	PROC WELD_20s_ALL()
        ActUnit STN1;
	    AccSet 75, 75;
	    MoveJ pjthomeSTA1zero, vCellSpeed, fine, tWeldGun\WObj:=wobj0;
        TPErase;
        !UNtilt19;
        TPWrite "NOW SEARCHING THE FIRST HALF OF WELD 'G'";
		GOTO GPOINT1stHALF;
        !!!!THIS IS THE ENTIRE "G" Search in Position EDIT STRING IN CORRECT ORDER!!!!
		PDispOff;
		MoveJ G19air2, vExtMax, z1, tWeldGun\WObj:=wobjHsideplate;
		MoveL RelTool(YG19S,0,-100,-150), v500, z1, tWeldGun\WObj:=wobjHsideplate;
		Search_1D SR_YZ_TEMP\SearchStop:=YZ_Temp, YG19S, YG19E, v300, tWeldGun\WObj:=wobjHsideplate\SchSpeed:=10;
         GHLM_YZ_POINT_SETTER G19, YZ_Temp, AA19;
        TPWrite "SRG19 XYZ:="\Pos:=SR_YZ_TEMP.trans;
		MoveL RelTool(YG19S,0,0,0), v500, z1, tWeldGun\WObj:=wobjHsideplate;
		Search_1D SR_YZ_TEMP\SearchStop:=YZ_Temp, YG15S, YG15E, v300, tWeldGun\WObj:=wobjHsideplate\SchSpeed:=10;
         GHLM_YZ_POINT_SETTER G15, YZ_Temp, AA15;
        TPWrite "SRG15 XYZ:="\Pos:=SR_YZ_TEMP.trans;
		MoveL RelTool(YG15S,0,0,0), v500, z1, tWeldGun\WObj:=wobjHsideplate;
		Search_1D SR_YZ_TEMP\SearchStop:=YZ_Temp, YG21S, YG21E, v300, tWeldGun\WObj:=wobjHsideplate\SchSpeed:=10;
         GHLM_YZ_POINT_SETTER G21, YZ_Temp, AA21;
        TPWrite "SRG21 XYZ:="\Pos:=SR_YZ_TEMP.trans;
		MoveL RelTool(YG21S,0,0,0), v500, z1, tWeldGun\WObj:=wobjHsideplate;
		Search_1D SR_YZ_TEMP\SearchStop:=YZ_Temp, YG0S, YG0E, v300, tWeldGun\WObj:=wobjHsideplate\SchSpeed:=10;
         GHLM_YZ_POINT_SETTER G0, YZ_Temp, AA0;
        TPWrite "SRG0 XYZ:="\Pos:=SR_YZ_TEMP.trans;
		MoveL RelTool(YG0S,0,0,0), v500, z1, tWeldGun\WObj:=wobjHsideplate;
		Search_1D SR_YZ_TEMP\SearchStop:=YZ_Temp, YG25S, YG25E, v300, tWeldGun\WObj:=wobjHsideplate\SchSpeed:=10;
         GHLM_YZ_POINT_SETTER G25, YZ_Temp, AA25;
        TPWrite "SRG25 XYZ:="\Pos:=SR_YZ_TEMP.trans;
		MoveL RelTool(YG25S,0,0,0), v500, z1, tWeldGun\WObj:=wobjHsideplate;
		Search_1D SR_YZ_TEMP\SearchStop:=YZ_Temp, YG29S, YG29E, v300, tWeldGun\WObj:=wobjHsideplate\SchSpeed:=10;
         GHLM_YZ_POINT_SETTER G29, YZ_Temp, AA29;
        TPWrite "SRG29 XYZ:="\Pos:=SR_YZ_TEMP.trans;
		MoveL RelTool(YG29S,0,0,0), v500, z1, tWeldGun\WObj:=wobjHsideplate;
		MoveJ G29air3, vExtMax, z1, tWeldGun\WObj:=wobjHsideplate;
        SEARCH_Gx;
        SET_G20s_X;
		PDispOff;
		MoveJ G19air1, vExtMax, z1, tWeldGun\WObj:=wobjHsideplate;
		MoveJ RelTool(G195L,0,-50,-50), v300, z1, tWeldGun\WObj:=wobjHtip;
		MoveL G195L, v100, z1, tWeldGun\WObj:=wobjHtip;
		MoveL G195, v100, z1, tWeldGun\WObj:=wobjHtip;
		MoveL G19, v100, z1, tWeldGun\WObj:=wobjHsideplate;
		MoveL RelTool(G15,0,0,-15), v100, z1, tWeldGun\WObj:=wobjHsideplate;
		MoveL G15, v100, z1, tWeldGun\WObj:=wobjHsideplate;
		MoveL RelTool(G21,0,0,-15), v100, z1, tWeldGun\WObj:=wobjHsideplate;
		MoveL G21, v100, z1, tWeldGun\WObj:=wobjHsideplate;
		MoveL RelTool(G21,0,0,-15), v100, z1, tWeldGun\WObj:=wobjHsideplate;
		MoveL G0, v100, z1, tWeldGun\WObj:=wobjHsideplate;
		MoveL RelTool(G0,0,0,-15), v100, z1, tWeldGun\WObj:=wobjHsideplate;
		MoveL RelTool(G25,0,0,-15), v100, z1, tWeldGun\WObj:=wobjHsideplate;
		MoveL G25, v100, z1, tWeldGun\WObj:=wobjHsideplate;
		MoveL RelTool(G25,0,0,-150), v100, z1, tWeldGun\WObj:=wobjHsideplate;
		MoveL G29, v100, z1, tWeldGun\WObj:=wobjHsideplate;
		MoveL RelTool(G29,0,0,-150), v100, z1, tWeldGun\WObj:=wobjHsideplate;
		MoveL RelTool(G0,0,0,-150), v100, z1, tWeldGun\WObj:=wobjHsideplate;
        !!  IF THIS IS AN H ARM THEN WE WILL RUN 1_THRU_8
        !!  IF THIS IS A G ARM THEN WE WILL RUN THE CAM-SIDE WELDS
		PDispOff;
         SET_G20s_X;
		MoveJ RelTool(G195L,0,-150,-150), v300, z1, tWeldGun\WObj:=wobjHtip;
        GOTO GWELDFIRST;
        GPOINT1stHALF:
        !!!!GETTING IN POSITION FOR THE FIRST 3 Y SEARCHES ON THE G WELD
        PDispOff;
		MoveJ G19air1, vExtMax, z1, tWeldGun\WObj:=wobjHsideplate;
		MoveL RelTool(YG19S,0,-100,-150), v500, z1, tWeldGun\WObj:=wobjHsideplate;
		Search_1D SR_YZ_TEMP\SearchStop:=YZ_Temp, YG19S, YG19E, v300, tWeldGun\WObj:=wobjHsideplate\SchSpeed:=10;
         GHLM_YZ_POINT_SETTER G19, YZ_Temp, AA19;
        TPWrite "SRG19 XYZ:="\Pos:=SR_YZ_TEMP.trans;
		MoveL RelTool(YG19S,0,0,0), v500, z1, tWeldGun\WObj:=wobjHsideplate;
		Search_1D SR_YZ_TEMP\SearchStop:=YZ_Temp, YG15S, YG15E, v300, tWeldGun\WObj:=wobjHsideplate\SchSpeed:=10;
         GHLM_YZ_POINT_SETTER G15, YZ_Temp, AA15;
        TPWrite "SRG15 XYZ:="\Pos:=SR_YZ_TEMP.trans;
		MoveL RelTool(YG15S,0,0,0), v500, z1, tWeldGun\WObj:=wobjHsideplate;
		Search_1D SR_YZ_TEMP\SearchStop:=YZ_Temp, YG21S, YG21E, v300, tWeldGun\WObj:=wobjHsideplate\SchSpeed:=10;
         GHLM_YZ_POINT_SETTER G21, YZ_Temp, AA21;
        TPWrite "SRG21 XYZ:="\Pos:=SR_YZ_TEMP.trans;
		MoveL RelTool(YG21S,0,0,0), v500, z1, tWeldGun\WObj:=wobjHsideplate;
		MoveL RelTool(YG21S,0,-100,0), v500, z1, tWeldGun\WObj:=wobjHsideplate;
 		MoveJ G19air1, vExtMax, z1, tWeldGun\WObj:=wobjHsideplate;
        SEARCH_Gx;
        SET_G20s_X;
		MoveJ G19air1, vExtMax, z1, tWeldGun\WObj:=wobjHsideplate;
		MoveJ RelTool(G195L,0,-50,-150), vExtMax, z1, tWeldGun\WObj:=wobjHtip;
        GWELDFIRST:
        IF bWO458only = TRUE OR bWO459only = TRUE THEN
        dripstop_G;
        ENDIF
        TPWrite "NOW WELDING THE FIRST THIRD OF WELD 'G'";
		MoveL RelTool(G195L,0,-50,-150), vExtMax, z1, tWeldGun\WObj:=wobjHtip;
		ArcLStart G195L, v100, smGH29, wdGH29\Weave:=wvGH29, fine, tWeldGun\WObj:=wobjHtip\Track:=trGHTBR;
		ArcL G195, v100, smGH29, wdGH29\Weave:=wvGH29, z1, tWeldGun\WObj:=wobjHtip\Track:=trGHTBR;
		ArcCEnd G15, G21, v100, smGH29, wdGH29\Weave:=wvGH29, fine, tWeldGun\WObj:=wobjHsideplate\Track:=trGHTBR;
		MoveL RelTool(G21,0,0,-150), vExtMax, z1, tWeldGun\WObj:=wobjHsideplate;
		MoveJ RelTool(G21,0,0,-200), vExtMax, z1, tWeldGun\WObj:=wobjHsideplate;
		MoveJ pjthomeSTA1zero, vCellSpeed, fine, tWeldGun\WObj:=wobj0;
        !!GOING TO THE H SIDE!!!
           MoveJ RelTool(H21,0,0,-500), vExtMax, z1, tWeldGun\WObj:=wobjHsideplate;
        TPErase;
        TPWrite "NOW WORKING ON FIRST HALF OF WELD 'H'";
		GOTO HPOINT1stHALF;
        !!!!THIS IS THE ENTIRE "H" SEARCHES EDIT STRING IN CORRECT ORDER!!!!
		PDispOff;
		MoveJ H19air1, vExtMax, z1, tWeldGun\WObj:=wobjHsideplate;
		MoveL RelTool(YH19S,150,70,-150), v500, z1, tWeldGun\WObj:=wobjHsideplate;
		Search_1D SR_YZ_TEMP\SearchStop:=YZ_Temp, YH19S, YH19E, v300, tWeldGun\WObj:=wobjHsideplate\SchSpeed:=10;
         GHLM_YZ_POINT_SETTER H19, YZ_Temp, AA19;
        TPWrite "SRH19 XYZ:="\Pos:=SR_YZ_TEMP.trans;
		MoveL RelTool(YH19S,0,0,0), v500, z1, tWeldGun\WObj:=wobjHsideplate;
		Search_1D SR_YZ_TEMP\SearchStop:=YZ_Temp, YH15S, YH15E, v300, tWeldGun\WObj:=wobjHsideplate\SchSpeed:=10;
         GHLM_YZ_POINT_SETTER H15, YZ_Temp, AA15;
        TPWrite "SRH15 XYZ:="\Pos:=SR_YZ_TEMP.trans;
		MoveL RelTool(YH15S,0,0,0), v500, z1, tWeldGun\WObj:=wobjHsideplate;
		Search_1D SR_YZ_TEMP\SearchStop:=YZ_Temp, YH21S, YH21E, v300, tWeldGun\WObj:=wobjHsideplate\SchSpeed:=10;
         GHLM_YZ_POINT_SETTER H21, YZ_Temp, AA21;
        TPWrite "SRH21 XYZ:="\Pos:=SR_YZ_TEMP.trans;
		MoveL RelTool(YH21S,0,0,0), v500, z1, tWeldGun\WObj:=wobjHsideplate;
		Search_1D SR_YZ_TEMP\SearchStop:=YZ_Temp, YH0S, YH0E, v300, tWeldGun\WObj:=wobjHsideplate\SchSpeed:=10;
         GHLM_YZ_POINT_SETTER H0, YZ_Temp, AA0;
        TPWrite "SRH0 XYZ:="\Pos:=SR_YZ_TEMP.trans;
		MoveL RelTool(YH0S,0,0,0), v500, z1, tWeldGun\WObj:=wobjHsideplate;
		Search_1D SR_YZ_TEMP\SearchStop:=YZ_Temp, YH25S, YH25E, v300, tWeldGun\WObj:=wobjHsideplate\SchSpeed:=10;
         GHLM_YZ_POINT_SETTER H25, YZ_Temp, AA25;
        TPWrite "SRH25 XYZ:="\Pos:=SR_YZ_TEMP.trans;
		MoveL RelTool(YH25S,0,0,0), v500, z1, tWeldGun\WObj:=wobjHsideplate;
		Search_1D SR_YZ_TEMP\SearchStop:=YZ_Temp, YH29S, YH29E, v300, tWeldGun\WObj:=wobjHsideplate\SchSpeed:=10;
         GHLM_YZ_POINT_SETTER H29, YZ_Temp, AA29;
        TPWrite "SRH29 XYZ:="\Pos:=SR_YZ_TEMP.trans;
		MoveL RelTool(YH29S,0,0,0), v500, z1, tWeldGun\WObj:=wobjHsideplate;
		MoveL RelTool(YH29S,100,100,0), v500, z1, tWeldGun\WObj:=wobjHsideplate;
		MoveJ H29air1, vExtMax, z1, tWeldGun\WObj:=wobjHsideplate;
        SEARCH_Hx;
        SET_H20s_X;
		MoveJ H19air1, vExtMax, z1, tWeldGun\WObj:=wobjHsideplate;
		MoveJ RelTool(H19,0,-100,-250), vExtMax, z1, tWeldGun\WObj:=wobjHsideplate;
		MoveL RelTool(H195L,0,-50,-50), v300, z1, tWeldGun\WObj:=wobjHtip;
        !!!!THIS IS THE ENTIRE "H" BASEPOINTS EDIT STRING IN CORRECT ORDER!!!!
		MoveL H195L, v100, z1, tWeldGun\WObj:=wobjHtip;
		MoveL H195, v100, z1, tWeldGun\WObj:=wobjHtip;
		MoveL H19, v100, z1, tWeldGun\WObj:=wobjHsideplate;
		MoveL RelTool(H15,0,0,-15), v100, z1, tWeldGun\WObj:=wobjHsideplate;
		MoveL H15, v100, z1, tWeldGun\WObj:=wobjHsideplate;
		MoveL RelTool(H21,0,0,-15), v100, z1, tWeldGun\WObj:=wobjHsideplate;
		MoveL H21, v100, z1, tWeldGun\WObj:=wobjHsideplate;
		MoveL RelTool(H0,0,0,-35), v100, z1, tWeldGun\WObj:=wobjHsideplate;
		MoveL H0, v100, z1, tWeldGun\WObj:=wobjHsideplate;
		MoveL RelTool(H25,0,0,-15), v100, z1, tWeldGun\WObj:=wobjHsideplate;
		MoveL H25, v100, z1, tWeldGun\WObj:=wobjHsideplate;
		MoveL RelTool(H25,0,0,-15), v100, z1, tWeldGun\WObj:=wobjHsideplate;
		MoveL H29, v100, z1, tWeldGun\WObj:=wobjHsideplate;
		MoveL RelTool(H29,0,0,-150), v100, z1, tWeldGun\WObj:=wobjHsideplate;
		MoveL RelTool(H0,0,0,-150), v100, z1, tWeldGun\WObj:=wobjHsideplate;
		PDispOff;
        PDispOff;
        SET_H20s_X;
		MoveJ RelTool(H195L,0,-150,-150), v300, z1, tWeldGun\WObj:=wobjHtip;
        GOTO HWELDSFIRSThalf;
        HPOINT1stHALF:
		PDispOff;
        !!!!GETTING IN POSITION FOR THE FIRST 3 Y SEARCHES ON THE H WELD
		MoveJ H19air1, vExtMax, z1, tWeldGun\WObj:=wobjHsideplate;
		MoveL RelTool(YH19S,150,70,-150), v500, z1, tWeldGun\WObj:=wobjHsideplate;
		Search_1D SR_YZ_TEMP\SearchStop:=YZ_Temp, YH19S, YH19E, v300, tWeldGun\WObj:=wobjHsideplate\SchSpeed:=10;
         GHLM_YZ_POINT_SETTER H19, YZ_Temp, AA19;
        TPWrite "SRH19 XYZ:="\Pos:=SR_YZ_TEMP.trans;
		MoveL RelTool(YH19S,0,0,0), v500, z1, tWeldGun\WObj:=wobjHsideplate;
		Search_1D SR_YZ_TEMP\SearchStop:=YZ_Temp, YH15S, YH15E, v300, tWeldGun\WObj:=wobjHsideplate\SchSpeed:=10;
         GHLM_YZ_POINT_SETTER H15, YZ_Temp, AA15;
        TPWrite "SRH15 XYZ:="\Pos:=SR_YZ_TEMP.trans;
		MoveL RelTool(YH15S,0,0,0), v500, z1, tWeldGun\WObj:=wobjHsideplate;
		Search_1D SR_YZ_TEMP\SearchStop:=YZ_Temp, YH21S, YH21E, v300, tWeldGun\WObj:=wobjHsideplate\SchSpeed:=10;
         GHLM_YZ_POINT_SETTER H21, YZ_Temp, AA21;
        TPWrite "SRH21 XYZ:="\Pos:=SR_YZ_TEMP.trans;
		MoveL RelTool(YH21S,0,0,0), v500, z1, tWeldGun\WObj:=wobjHsideplate;
		MoveL RelTool(YH21S,100,100,-150), v500, z1, tWeldGun\WObj:=wobjHsideplate;
        !!!!GETTING IN POSITION FOR THE FIRST 2 X SEARCHES ON THE H WELD
		MoveJ H19air1, vExtMax, z1, tWeldGun\WObj:=wobjHsideplate;
		MoveJ H19air10, vExtMax, z1, tWeldGun\WObj:=wobjHsideplate;
        SEARCH_Hx;
        SET_H20s_X;
        MoveJ H19air10, vExtMax, z1, tWeldGun\WObj:=wobjHsideplate;
		MoveJ H19air1, vExtMax, z1, tWeldGun\WObj:=wobjHsideplate;
		MoveJ RelTool(H195L,0,-40,-100), vExtMax, z1, tWeldGun\WObj:=wobjHtip;
        HWELDSFIRSThalf:
		MoveL RelTool(H195L,0,-20,-50), vExtMax, z1, tWeldGun\WObj:=wobjHtip;
		ArcLStart H195L, v100, smGH29, wdGH29\Weave:=wvGH29, fine, tWeldGun\WObj:=wobjHtip\Track:=trGH;
		ArcL H195, v100, smGH29, wdGH29\Weave:=wvGH29, z1, tWeldGun\WObj:=wobjHtip\Track:=trGH;
		ArcCEnd H15, H21, v100, smGH29, wdGH29\Weave:=wvGH29, fine, tWeldGun\WObj:=wobjHsideplate\Track:=trGH;
		MoveL RelTool(H21,0,0,-50), v300, z1, tWeldGun\WObj:=wobjHsideplate;
        TPErase;
		MoveL RelTool(H21,0,0,-500), vExtMax, z5, tWeldGun\WObj:=wobjHsideplate;
		MoveJ pjthomeSTA1zero, vCellSpeed, fine, tWeldGun\WObj:=wobj0;
        TPErase;
        TPWrite "NOW WORKING ON LAST HALF OF WELD 'G'";
		MoveJ RelTool(YG29S,0,-100,-150), vExtMax, z1, tWeldGun\WObj:=wobjHsideplate;
		Search_1D SR_YZ_TEMP\SearchStop:=YZ_Temp, YG29S, YG29E, v300, tWeldGun\WObj:=wobjHsideplate\SchSpeed:=10;
         GHLM_YZ_POINT_SETTER G29, YZ_Temp, AA29;
        TPWrite "SRG29 XYZ:="\Pos:=SR_YZ_TEMP.trans;
		MoveL RelTool(YG29S,0,0,0), v500, z1, tWeldGun\WObj:=wobjHsideplate;
		Search_1D SR_YZ_TEMP\SearchStop:=YZ_Temp, YG25S, YG25E, v300, tWeldGun\WObj:=wobjHsideplate\SchSpeed:=10;
         GHLM_YZ_POINT_SETTER G25, YZ_Temp, AA25;
        TPWrite "SRG25 XYZ:="\Pos:=SR_YZ_TEMP.trans;
		MoveL RelTool(YG25S,0,0,0), v500, z1, tWeldGun\WObj:=wobjHsideplate;
		Search_1D SR_YZ_TEMP\SearchStop:=YZ_Temp, YG0S, YG0E, v300, tWeldGun\WObj:=wobjHsideplate\SchSpeed:=10;
         GHLM_YZ_POINT_SETTER G0, YZ_Temp, AA0;
        TPWrite "SRG0 XYZ:="\Pos:=SR_YZ_TEMP.trans;
		MoveL RelTool(YG0S,0,0,0), v500, z1, tWeldGun\WObj:=wobjHsideplate;
		MoveJ G29air3, vExtMax, z1, tWeldGun\WObj:=wobjHsideplate;
        SEARCH_Gx;
        SET_G20s_X;
		MoveJ G29air1, vExtMax, z1, tWeldGun\WObj:=wobjHsideplate;
        IF pivCAM = FALSE THEN
            PivGX18_Rnd Gx_weld_piv;
            WELD_ALLPIV_1thru8 "G";
    ! RESTART here IF the arm is an -"H"- style Pivot Catsing
            ArcLStart G_RND_7, v100, smGH29, wdGH29\Weave:=wvGH29, fine, tWeldGun\WObj:=wobj_PivCam\Track:=trGHTBL;
            GOTO QUIT_IFing_AROUND;
                ELSEIF pivCAM = TRUE THEN
            PivGX18_Cam_18_R1 Gx_weld_piv;
            Piv_side_Welds "G";
    ! RESTART here IF the arm is an -"F"- style Pivot Casting
        !Stop;
        IF bWO458only = TRUE OR bWO459only = TRUE THEN
        dripstop_G;
        ENDIF
		MoveL RelTool(GCam_SidePIV_S,0,0,-70), v500, z5, tWeldGun\WObj:=wobj_PivCam;
            ArcLStart GCam_SidePIV_S, v100, smGH29, wdGH29\Weave:=wvGH29, z1, tWeldGun\WObj:=wobj_PivCam\Track:=trGHTBL;
            ArcL GCam_SidePIV_Sm, v100, smGH29, wdGH29\Weave:=wvGH29, z1, tWeldGun\WObj:=wobj_PivCam\Track:=trGHTBL;
            ArcL GCam_SidePIV_E, v100, smGH29, wdGH29\Weave:=wvGH29, z1, tWeldGun\WObj:=wobj_PivCam\Track:=trGHTBL;
            GOTO QUIT_IFing_AROUND;
        ENDIF
        QUIT_IFing_AROUND:
        PDispOff;
		ArcL G29, v100, smGH29, wdGH29\Weave:=wvGH29, z1, tWeldGun\WObj:=wobjHsideplate\Track:=trGHTBL;
		ArcCEnd G25, G0, v100, smGH29, wdGH29\Weave:=wvGH29, fine, tWeldGun\WObj:=wobjHsideplate\Track:=trGHTBL;
		MoveJ RelTool(G0,0,0,-150), vExtMax, z1, tWeldGun\WObj:=wobjHsideplate;
		MoveJ pjthomeSTA1zero, vCellSpeed, z1, tWeldGun\WObj:=wobj0;
        TPErase;
        TPWrite "NOW SEARCHING AND WELDING THE LAST HALF OF WELD 'H'";
		MoveJ RelTool(H0,0,0,-500), vExtMax, z5, tWeldGun\WObj:=wobjHsideplate;
        !!!!GETTING IN POSITION FOR THE LAST 3 Y SEARCHES ON THE H WELD
		MoveJ H29air1, vExtMax, z1, tWeldGun\WObj:=wobjHsideplate;
		MoveL RelTool(YH29S,0,150,-150), v500, z1, tWeldGun\WObj:=wobjHsideplate;
		Search_1D SR_YZ_TEMP\SearchStop:=YZ_Temp, YH29S, YH29E, v300, tWeldGun\WObj:=wobjHsideplate\SchSpeed:=10;
         GHLM_YZ_POINT_SETTER H29, YZ_Temp, AA29;
        TPWrite "SRH29 XYZ:="\Pos:=SR_YZ_TEMP.trans;
		MoveL RelTool(YH29S,0,0,0), v500, z1, tWeldGun\WObj:=wobjHsideplate;
		Search_1D SR_YZ_TEMP\SearchStop:=YZ_Temp, YH25S, YH25E, v300, tWeldGun\WObj:=wobjHsideplate\SchSpeed:=10;
         GHLM_YZ_POINT_SETTER H25, YZ_Temp, AA25;
        TPWrite "SRH25 XYZ:="\Pos:=SR_YZ_TEMP.trans;
		MoveL RelTool(YH25S,0,0,0), v500, z1, tWeldGun\WObj:=wobjHsideplate;
		Search_1D SR_YZ_TEMP\SearchStop:=YZ_Temp, YH0S, YH0E, v300, tWeldGun\WObj:=wobjHsideplate\SchSpeed:=10;
         GHLM_YZ_POINT_SETTER H0, YZ_Temp, AA0;
        TPWrite "SRH0 XYZ:="\Pos:=SR_YZ_TEMP.trans;
		MoveL RelTool(YH0S,0,0,0), v500, z1, tWeldGun\WObj:=wobjHsideplate;
		MoveL RelTool(YH0S,100,100,-150), v500, z1, tWeldGun\WObj:=wobjHsideplate;
        !!!!GETTING IN POSITION FOR THE LAST 2 X SEARCHES ON THE H WELD
		MoveJ H29air1, vExtMax, z1, tWeldGun\WObj:=wobjHsideplate;
		MoveJ H29air12, vExtMax, z1, tWeldGun\WObj:=wobjHsideplate;
        SEARCH_Hx;
        SET_H20s_X;
		MoveJ H29air12, vExtMax, z1, tWeldGun\WObj:=wobjHsideplate;
        IF pivCAM = FALSE THEN
            PivHX18_Rnd Hx_weld_piv;
            WELD_ALLPIV_1thru8 "H";
    ! RESTART here IF the arm is an -"H"- style Pivor Catsing
    ArcLStart H_RND_7, v100, smGH29, wdGH29\Weave:=wvGH29, fine, tWeldGun\WObj:=wobj_PivCam\Track:=trGHTBL;
            GOTO QUIT_snIFing_AROUND;
           ELSEIF pivCAM = TRUE THEN
            PivHX18_Cam_18_R1 Hx_weld_piv;
            Piv_side_Welds "H";
    ! RESTART here IF the arm is an -"F"- style Pivot Casting
            ArcLStart HCam_SidePIV_S, v100, smGH29, wdGH29\Weave:=wvGH29, z1, tWeldGun\WObj:=wobj_PivCam\Track:=trGHTBL;
            ArcL HCam_SidePIV_Sm, v100, smGH29, wdGH29\Weave:=wvGH29, z1, tWeldGun\WObj:=wobj_PivCam\Track:=trGHTBL;
            ArcL HCam_SidePIV_E, v100, smGH29, wdGH29\Weave:=wvGH29, z1, tWeldGun\WObj:=wobj_PivCam\Track:=trGHTBL;
            GOTO QUIT_snIFing_AROUND;
        ENDIF
        QUIT_snIFing_AROUND:
		PDispOff;
		ArcL H29, v100, smGH29, wdGH29\Weave:=wvGH29, z1, tWeldGun\WObj:=wobjHsideplate\Track:=trGH;
		ArcCEnd H25, H0, v100, smGH29, wdGH29\Weave:=wvGH29, z1, tWeldGun\WObj:=wobjHsideplate\Track:=trGH;
		MoveL RelTool(H0,0,0,-150), vExtMax, z1, tWeldGun\WObj:=wobjHsideplate;
        TPErase;
        TPErase;
        TPWrite "DONE WELDING FRONT WRAPPER THE track bias WAY";
		MoveJ RelTool(H0,0,0,-500), vExtMax, z5, tWeldGun\WObj:=wobjHsideplate;
		MoveJ pjthomeSTA1zero, vCellSpeed, fine, tWeldGun\WObj:=wobj0;
		getout:
	ENDPROC

	PROC WELD_60s_ALL()
		ActUnit STN1;
	    AccSet 75, 75;
		MoveJ pjthomeSTA1zero, vCellSpeed, fine, tWeldGun\WObj:=wobj0;
        TPErase;
        TPWrite "NOW WORKING ON WELD 'L70 TO 67'";
		GOTO LPOINT70_67;
        !!!!!THIS IS THE EDIT STRING FOR L 60S searches IN ORDER
    	PDispOff;
		MoveJ YL69air1, vExtMax, z1, tWeldGun\WObj:=wobjHsideplate;
		MoveL YL69air2, vExtMax, z1, tWeldGun\WObj:=wobjHsideplate;
		MoveL Offs(YL69E,150,200,0), v500, z1, tWeldGun\WObj:=wobjHsideplate;
		MoveL RelTool(YL69S,0,0,0), v500, z1, tWeldGun\WObj:=wobjHsideplate;
		Search_1D SR_YZ_TEMP\SearchStop:=YZ_Temp, YL69S, YL69E, v300, tWeldGun\WObj:=wobjHsideplate\SchSpeed:=10;
        GHLM_YZ_POINT_SETTER L69, YZ_Temp, AA69;
        TPWrite "SRL69 XYZ:="\Pos:=SR_YZ_TEMP.trans;
		MoveL RelTool(YL69S,0,0,0), v500, z1, tWeldGun\WObj:=wobjHsideplate;
		Search_1D SR_YZ_TEMP\SearchStop:=YZ_Temp, YL67S, YL67E, v300, tWeldGun\WObj:=wobjHsideplate\SchSpeed:=10;
        GHLM_YZ_POINT_SETTER L67, YZ_Temp, AA67;
        TPWrite "SRL67 XYZ:="\Pos:=SR_YZ_TEMP.trans;
		MoveL RelTool(YL67S,0,0,0), v500, z1, tWeldGun\WObj:=wobjHsideplate;
		Search_1D SR_YZ_TEMP\SearchStop:=YZ_Temp, YL61S, YL61E, v300, tWeldGun\WObj:=wobjHsideplate\SchSpeed:=10;
        GHLM_YZ_POINT_SETTER L61, YZ_Temp, AA61;
        TPWrite "SRL61 XYZ:="\Pos:=SR_YZ_TEMP.trans;
		MoveL RelTool(YL61S,0,0,0), v500, z1, tWeldGun\WObj:=wobjHsideplate;
		MoveL RelTool(YL67S,-100,0,-50), v500, z1, tWeldGun\WObj:=wobjHsideplate;
		MoveL YL69air2, vExtMax, z1, tWeldGun\WObj:=wobjHsideplate;
		MoveJ halfwayhome_L, vExtMax, z1, tWeldGun\WObj:=wobjHsideplate;
        SEARCH_Lx;
        SET_L60s_X;
		MoveJ halfwayhome_L, vExtMax, z1, tWeldGun\WObj:=wobjHsideplate;
		MoveJ YL69air10, vExtMax, z1, tWeldGun\WObj:=wobjHsideplate;
		MoveJ YL69air1, vExtMax, z1, tWeldGun\WObj:=wobjHsideplate;
		MoveJ RelTool(L68,0,0,-400), vExtMax, z1, tWeldGun\WObj:=wobjHsideplate;
        !!!!!THIS IS THE EDIT STRING FOR L 60S BASEPOINTS
		PDispOff;
		MoveL RelTool(L69,0,0,-50), v100, z1, tWeldGun\WObj:=wobjHsideplate;
		MoveL L69, v100, z1, tWeldGun\WObj:=wobjHsideplate;
		MoveL RelTool(L67,0,0,-25), v100, z1, tWeldGun\WObj:=wobjHsideplate;
		MoveL L67, v100, z1, tWeldGun\WObj:=wobjHsideplate;
		MoveL RelTool(L67,0,0,-55), v100, z1, tWeldGun\WObj:=wobjHsideplate;
		MoveL RelTool(L61,0,0,-25), v100, z1, tWeldGun\WObj:=wobjHsideplate;
		MoveL L61, v100, z1, tWeldGun\WObj:=wobjHsideplate;
		MoveL RelTool(L61,0,0,-25), v100, z1, tWeldGun\WObj:=wobjHsideplate;
		MoveL RelTool(L67,0,0,-25), v100, z1, tWeldGun\WObj:=wobjHsideplate;
		PDispOff;
        SET_L60s_X;
		MoveL RelTool(L67,0,0,-325), v100, z1, tWeldGun\WObj:=wobjHsideplate;
        GOTO FIRSTTHIRDL;
        LPOINT70_67:
		MoveJ YL69air1, vExtMax, z1, tWeldGun\WObj:=wobjHsideplate;
		MoveL YL69air2, v500, z1, tWeldGun\WObj:=wobjHsideplate;
		MoveL Offs(YL69S,150,200,0), v500, z1, tWeldGun\WObj:=wobjHsideplate;
		MoveL RelTool(YL69S,0,0,0), v500, z1, tWeldGun\WObj:=wobjHsideplate;
		Search_1D SR_YZ_TEMP\SearchStop:=YZ_Temp, YL69S, YL69E, v300, tWeldGun\WObj:=wobjHsideplate\SchSpeed:=10;
        GHLM_YZ_POINT_SETTER L69, YZ_Temp, AA69;
        TPWrite "SRL69 XYZ:="\Pos:=SR_YZ_TEMP.trans;
		MoveL RelTool(YL69S,0,0,0), v500, z1, tWeldGun\WObj:=wobjHsideplate;
		Search_1D SR_YZ_TEMP\SearchStop:=YZ_Temp, YL67S, YL67E, v300, tWeldGun\WObj:=wobjHsideplate\SchSpeed:=10;
        GHLM_YZ_POINT_SETTER L67, YZ_Temp, AA67;
        TPWrite "SRL67 XYZ:="\Pos:=SR_YZ_TEMP.trans;
		MoveL RelTool(YL67S,0,0,0), v500, z1, tWeldGun\WObj:=wobjHsideplate;
		Search_1D SR_YZ_TEMP\SearchStop:=YZ_Temp, YL61S, YL61E, v300, tWeldGun\WObj:=wobjHsideplate\SchSpeed:=10;
        GHLM_YZ_POINT_SETTER L61, YZ_Temp, AA61;
        TPWrite "SRL61 XYZ:="\Pos:=SR_YZ_TEMP.trans;
		MoveL RelTool(YL61S,0,0,0), v500, z1, tWeldGun\WObj:=wobjHsideplate;
		MoveL RelTool(YL67S,0,0,0), v500, z1, tWeldGun\WObj:=wobjHsideplate;
		MoveL RelTool(YL67S,-100,0,0), v500, z1, tWeldGun\WObj:=wobjHsideplate;
		MoveL YL69air2, vExtMax, z1, tWeldGun\WObj:=wobjHsideplate;
		MoveJ halfwayhome_L, vExtMax, z1, tWeldGun\WObj:=wobjHsideplate;
        SEARCH_Lx;
        SET_L60s_X;
		MoveJ halfwayhome_L, vExtMax, z1, tWeldGun\WObj:=wobjHsideplate;
		MoveJ YL69air10, vExtMax, z1, tWeldGun\WObj:=wobjHsideplate;
		MoveJ YL69air1, vExtMax, z1, tWeldGun\WObj:=wobjHsideplate;
        FIRSTTHIRDL:
		MoveJ RelTool(L67,0,0,-400), vExtMax, z1, tWeldGun\WObj:=wobjHsideplate;
		ArcLStart RelTool(L69,0,3,-4), v100, smLM10, wdLM10\Weave:=wvLM10, fine, tWeldGun\WObj:=wobjHsideplate\Track:=trLM10;
		ArcL L67, v100, smLM10, wdLM10\Weave:=wvLM10, z5, tWeldGun\WObj:=wobjHsideplate\Track:=trLM10;
		ArcLEnd RelTool(L61,0,-6,-2), v100, smLM10, wdLM10\Weave:=wvLM10, z5, tWeldGun\WObj:=wobjHsideplate\Track:=trLM10;
		MoveL RelTool(L67,0,0,-80), v100, z1, tWeldGun\WObj:=wobjHsideplate;
		MoveJ RelTool(L67,0,0,-400), vExtMax, z1, tWeldGun\WObj:=wobjHsideplate;
        TPErase;
        TPWrite "NOW WORKING ON WELD 'M70 to 67'";
		GOTO MPOINT70_67;
        !!!!!THIS IS THE EDIT STRING FOR M 60S searches IN ORDER
    	PDispOff;
		MoveJ YM69air0, vExtMax, z1, tWeldGun\WObj:=wobjHsideplate;
		MoveJ YM69air1, vExtMax, z1, tWeldGun\WObj:=wobjHsideplate;
		MoveJ YM69air2, vExtMax, z1, tWeldGun\WObj:=wobjHsideplate;
		MoveL RelTool(YM69S,0,0,0), vExtMax, z1, tWeldGun\WObj:=wobjHsideplate;
		Search_1D SR_YZ_TEMP\SearchStop:=YZ_Temp, YM69S, YM69E, v300, tWeldGun\WObj:=wobjHsideplate\SchSpeed:=10;
        GHLM_YZ_POINT_SETTER M69, YZ_Temp, AA69;
        TPWrite "SRM69 XYZ:="\Pos:=SR_YZ_TEMP.trans;
		MoveL RelTool(YM69S,0,0,0), v500, z1, tWeldGun\WObj:=wobjHsideplate;
		Search_1D SR_YZ_TEMP\SearchStop:=YZ_Temp, YM67S, YM67E, v300, tWeldGun\WObj:=wobjHsideplate\SchSpeed:=10;
        GHLM_YZ_POINT_SETTER M67, YZ_Temp, AA67;
        TPWrite "SRM67 XYZ:="\Pos:=SR_YZ_TEMP.trans;
		MoveL RelTool(YM67S,0,0,0), v500, z1, tWeldGun\WObj:=wobjHsideplate;
		Search_1D SR_YZ_TEMP\SearchStop:=YZ_Temp, YM61S, YM61E, v300, tWeldGun\WObj:=wobjHsideplate\SchSpeed:=10;
        GHLM_YZ_POINT_SETTER M61, YZ_Temp, AA61;
        TPWrite "SRM61 XYZ:="\Pos:=SR_YZ_TEMP.trans;
		MoveL RelTool(YM61S,0,0,0), v500, z1, tWeldGun\WObj:=wobjHsideplate;
		MoveL RelTool(YM61S,50,0,-60), v500, z1, tWeldGun\WObj:=wobjHsideplate;
		MoveJ YM69air2, vExtMax, z1, tWeldGun\WObj:=wobjHsideplate;
		MoveJ YM69air1, vExtMax, z1, tWeldGun\WObj:=wobjHsideplate;
		MoveJ halfwayhome_M, vExtMax, z1, tWeldGun\WObj:=wobjHsideplate;
        SEARCH_Mx;
        SET_M60s_X;
		MoveJ halfwayhome_M, vExtMax, z1, tWeldGun\WObj:=wobjHsideplate;
		MoveJ RelTool(M69,0,0,-450), vExtMax, z1, tWeldGun\WObj:=wobjHsideplate;
        !!!!!THIS IS THE EDIT STRING FOR M 60S BASEPOINTS
		PDispOff;
		MoveL RelTool(M69,0,0,-100), vExtMax, z1, tWeldGun\WObj:=wobjHsideplate;
		!sure to crash
		MoveL M69, v100, z1, tWeldGun\WObj:=wobjHsideplate;
		MoveL RelTool(M67,0,0,-25), v100, z1, tWeldGun\WObj:=wobjHsideplate;
		MoveL M67, v100, z1, tWeldGun\WObj:=wobjHsideplate;
		MoveL RelTool(M67,0,0,-55), v100, z1, tWeldGun\WObj:=wobjHsideplate;
		MoveL RelTool(M61,0,0,-25), v100, z1, tWeldGun\WObj:=wobjHsideplate;
		MoveL M61, v100, z1, tWeldGun\WObj:=wobjHsideplate;
		MoveL RelTool(M61,0,0,-25), v100, z1, tWeldGun\WObj:=wobjHsideplate;
		MoveL RelTool(M67,0,0,-450), vExtMax, z1, tWeldGun\WObj:=wobjHsideplate;
		MoveL RelTool(M69,0,0,-450), vExtMax, z1, tWeldGun\WObj:=wobjHsideplate;
		PDispOff;
        SET_M60s_X;
        GOTO FIRSTandLASTM;
        MPOINT70_67:
    	PDispOff;
		MoveJ YM69air0, vExtMax, z1, tWeldGun\WObj:=wobjHsideplate;
		MoveJ YM69air1, vExtMax, z1, tWeldGun\WObj:=wobjHsideplate;
		MoveJ YM69air2, vExtMax, z1, tWeldGun\WObj:=wobjHsideplate;
		MoveL RelTool(YM69S,0,0,0), vExtMax, z1, tWeldGun\WObj:=wobjHsideplate;
		Search_1D SR_YZ_TEMP\SearchStop:=YZ_Temp, YM69S, YM69E, v300, tWeldGun\WObj:=wobjHsideplate\SchSpeed:=10;
        GHLM_YZ_POINT_SETTER M69, YZ_Temp, AA69;
        TPWrite "SRM69 XYZ:="\Pos:=SR_YZ_TEMP.trans;
		MoveL RelTool(YM69S,0,0,0), v500, z1, tWeldGun\WObj:=wobjHsideplate;
		Search_1D SR_YZ_TEMP\SearchStop:=YZ_Temp, YM67S, YM67E, v300, tWeldGun\WObj:=wobjHsideplate\SchSpeed:=10;
        GHLM_YZ_POINT_SETTER M67, YZ_Temp, AA67;
        TPWrite "SRM67 XYZ:="\Pos:=SR_YZ_TEMP.trans;
		MoveL RelTool(YM67S,0,0,0), v500, z1, tWeldGun\WObj:=wobjHsideplate;
		Search_1D SR_YZ_TEMP\SearchStop:=YZ_Temp, YM61S, YM61E, v300, tWeldGun\WObj:=wobjHsideplate\SchSpeed:=10;
        GHLM_YZ_POINT_SETTER M61, YZ_Temp, AA61;
        TPWrite "SRM61 XYZ:="\Pos:=SR_YZ_TEMP.trans;
		MoveL RelTool(YM61S,0,0,0), v500, z1, tWeldGun\WObj:=wobjHsideplate;
		MoveL RelTool(YM67S,0,0,0), v500, z1, tWeldGun\WObj:=wobjHsideplate;
		MoveJ YM69air2, vExtMax, z1, tWeldGun\WObj:=wobjHsideplate;
		MoveJ YM69air1, vExtMax, z1, tWeldGun\WObj:=wobjHsideplate;
		MoveJ YM69air0, vExtMax, z1, tWeldGun\WObj:=wobjHsideplate;
		MoveJ halfwayhome_M, vExtMax, z1, tWeldGun\WObj:=wobjHsideplate;
        SEARCH_Mx;
        SET_M60s_X;
		MoveJ halfwayhome_M, vExtMax, z1, tWeldGun\WObj:=wobjHsideplate;
		MoveJ RelTool(M69,0,0,-450), vExtMax, z1, tWeldGun\WObj:=wobjHsideplate;
        FIRSTandLASTM:
		MoveL RelTool(M69,0,0,-100), v200, z1, tWeldGun\WObj:=wobjHsideplate;
		ArcLStart RelTool(M69,-3,0,-4), v100, smLM10, wdLM10\Weave:=wvLM10, fine, tWeldGun\WObj:=wobjHsideplate\Track:=trLM10;
		ArcL M67, v100, smLM10, wdLM10\Weave:=wvLM10, z5, tWeldGun\WObj:=wobjHsideplate\Track:=trLM10;
		ArcLEnd RelTool(M61,5,0,-2), v100, smLM10, wdLM10\Weave:=wvLM10, z5, tWeldGun\WObj:=wobjHsideplate\Track:=trLM10;
		MoveL RelTool(M67,0,0,-20), v100, z1, tWeldGun\WObj:=wobjHsideplate;
		MoveL RelTool(M67,0,0,-200), v100, z1, tWeldGun\WObj:=wobjHsideplate;
		MoveJ Offs(M67,250,-250,0), vExtMax, z5, tWeldGun\WObj:=wobjHsideplate;
        TPErase;
		MoveJ pjthomeSTA1zero, vCellSpeed, fine, tWeldGun\WObj:=wobj0;
        stepthru:
	ENDPROC

	PROC SEARCH_Ax()
		MoveJ halfwayhome_A, vExtMax, z1, tWeldGun\WObj:=wobjHsideplate;
		MoveL Offs(XA39E,100,0,0), vExtMax, z1, tWeldGun\WObj:=wobjHtip;
		Search_1D SRA39X\SearchStop:=X_Temp, Offs(XA39E,50,0,0), XA39E, v300, tWeldGun\WObj:=wobjHtip\SchSpeed:=10;
 		MoveL X_Temp, v50, fine, tWeldGun\WObj:=wobjHtip;
        WaitTime\InPos, 0.2;
		Ax_weld_tip := CRobT(\Tool:=tWeldGun\WObj:=wobjHsideplate);
        TPWrite "SRA39X XYZ:="\Pos:=SRA39X.trans;
		MoveL Offs(XA39E,100,0,0), v500, z1, tWeldGun\WObj:=wobjHtip;
		MoveL Offs(XA33E,100,0,0), v500, z1, tWeldGun\WObj:=wobjHanchor;
		Search_1D SRA33X\SearchStop:=X_Temp, Offs(XA33E,50,0,0), XA33E, v300, tWeldGun\WObj:=wobjHanchor\SchSpeed:=10;
 		MoveL X_Temp, v50, fine, tWeldGun\WObj:=wobjHanchor;
        WaitTime\InPos, 0.2;
		Ax_weld_anchor := CRobT(\Tool:=tWeldGun\WObj:=wobjHsideplate);
        TPWrite "SRA33X XYZ:="\Pos:=SRA33X.trans;
		MoveL Offs(XA33E,100,0,0), v500, z1, tWeldGun\WObj:=wobjHanchor;
		MoveL Offs(XA30E,100,0,0), v500, z1, tWeldGun\WObj:=wobjHanchor;
		Search_1D SRA30X\SearchStop:=X_Temp, Offs(XA30E,50,0,0), XA30E, v300, tWeldGun\WObj:=wobjHanchor\SchSpeed:=10;
 		MoveL X_Temp, v50, fine, tWeldGun\WObj:=wobjHanchor;
        WaitTime\InPos, 0.2;
		Ax_weld_piv := CRobT(\Tool:=tWeldGun\WObj:=wobjHsideplate);
        TPWrite "SRA30X XYZ:="\Pos:=SRA30X.trans;
		MoveL Offs(XA30E,150,100,0), v500, z1, tWeldGun\WObj:=wobjHanchor;
		MoveJ halfwayhome_A, vExtMax, z1, tWeldGun\WObj:=wobjHsideplate;
        BACK2A:
	ENDPROC

	PROC SEARCH_Bx()
		MoveJ halfwayhome_B, vExtMax, z1, tWeldGun\WObj:=wobjHsideplate;
		MoveL Offs(XB39E,-90,0,0), v500, z1, tWeldGun\WObj:=wobjHtip;
		Search_1D SRB39X\SearchStop:=X_Temp, Offs(XB39E,-50,0,0), XB39E, v300, tWeldGun\WObj:=wobjHtip\SchSpeed:=10;
 		MoveL X_Temp, v50, fine, tWeldGun\WObj:=wobjHtip;
        WaitTime\InPos, .1;
		Bx_weld_tip := CRobT(\Tool:=tWeldGun\WObj:=wobjHsideplate);
        TPWrite "SRB39X XYZ:="\Pos:=SRB39X.trans;
		MoveL Offs(XB39E,-90,0,0), v500, z1, tWeldGun\WObj:=wobjHtip;
		MoveL Offs(XB33E,-90,0,0), v500, z1, tWeldGun\WObj:=wobjHanchor;
		Search_1D SRB33X\SearchStop:=X_Temp, Offs(XB33E,-50,0,0), XB33E, v300, tWeldGun\WObj:=wobjHanchor\SchSpeed:=10;
 		MoveL X_Temp, v50, fine, tWeldGun\WObj:=wobjHanchor;
        WaitTime\InPos, .1;
		Bx_weld_anchor := CRobT(\Tool:=tWeldGun\WObj:=wobjHsideplate);
        TPWrite "SRB33X XYZ:="\Pos:=SRB33X.trans;
		MoveL Offs(XB33E,-90,0,0), v500, z1, tWeldGun\WObj:=wobjHanchor;
		MoveL Offs(XB30E,-90,0,0), v300, z1, tWeldGun\WObj:=wobjHanchor;
		Search_1D SRB30X\SearchStop:=X_Temp, Offs(XB30E,-50,0,0), XB30E, v300, tWeldGun\WObj:=wobjHanchor\SchSpeed:=10;
 		MoveL X_Temp, v50, fine, tWeldGun\WObj:=wobjHanchor;
        WaitTime\InPos, .1;
		Bx_weld_piv := CRobT(\Tool:=tWeldGun\WObj:=wobjHsideplate);
        TPWrite "SRB30X XYZ:="\Pos:=SRB30X.trans;
		MoveL Offs(XB30E,-90,0,0), v300, z1, tWeldGun\WObj:=wobjHanchor;
		MoveJ halfwayhome_B, vExtMax, z1, tWeldGun\WObj:=wobjHsideplate;
        BACK2B:
	ENDPROC

	PROC SEARCH_Gx()
		MoveJ halfwayhome_G, vExtMax, z1, tWeldGun\WObj:=wobjHsideplate;
		MoveJ Offs(XG29E,-100,0,0), v500, z1, tWeldGun\WObj:=wobjHpivot;
		Search_1D SRG29X\SearchStop:=X_Temp, Offs(XG29E,-50,0,0), XG29E, v300, tWeldGun\WObj:=wobjHpivot\SchSpeed:=10;
		MoveL X_Temp, v50, fine, tWeldGun\WObj:=wobjHpivot;
        WaitTime\InPos, .1;
		Gx_weld_piv := CRobT(\Tool:=tWeldGun\WObj:=wobjHsideplate);
        TPWrite "SRG29X XYZ:="\Pos:=SRG29X.trans;
		MoveL Offs(XG29E,-100,0,0), v500, z1, tWeldGun\WObj:=wobjHpivot;
		MoveJ Offs(XG0E,-100,0,0), v500, z1, tWeldGun\WObj:=wobjHanchor;
		Search_1D SRG0X\SearchStop:=X_Temp, Offs(XG0E,-50,0,0), XG0E, v300, tWeldGun\WObj:=wobjHanchor\SchSpeed:=10;
		MoveL X_Temp, v50, fine, tWeldGun\WObj:=wobjHanchor;
        WaitTime\InPos, .1;
		Gx_weld_anchor := CRobT(\Tool:=tWeldGun\WObj:=wobjHsideplate);
        TPWrite "SRG0X XYZ:="\Pos:=SRG0X.trans;
		MoveJ Offs(XG0E,-100,0,0), v500, z1, tWeldGun\WObj:=wobjHanchor;
		MoveJ Offs(XG19E,-100,0,0), v500, z1, tWeldGun\WObj:=wobjHtip;
		Search_1D SRG19X\SearchStop:=X_Temp, Offs(XG19E,-50,0,0), XG19E, v300, tWeldGun\WObj:=wobjHtip\SchSpeed:=10;
 		MoveL X_Temp, v50, fine, tWeldGun\WObj:=wobjHtip;
        WaitTime\InPos, .1;
		Gx_weld_tip := CRobT(\Tool:=tWeldGun\WObj:=wobjHsideplate);
        TPWrite "SRG19X XYZ:="\Pos:=SRG19X.trans;
		MoveJ Offs(XG19E,-200,0,0), v500, z1, tWeldGun\WObj:=wobjHtip;
        BACK2G:
	ENDPROC

	PROC SEARCH_Hx()
		MoveJ halfwayhome_H, vExtMax, z1, tWeldGun\WObj:=wobjHsideplate;
		MoveL Offs(XH29E,80,0,0), v500, z1, tWeldGun\WObj:=wobjHpivot;
		Search_1D SRH29X\SearchStop:=X_Temp, Offs(XH29E,50,0,0), XH29E, v300, tWeldGun\WObj:=wobjHpivot\SchSpeed:=10;
		MoveL X_Temp, v50, fine, tWeldGun\WObj:=wobjHpivot;
        WaitTime\InPos, .1;
		Hx_weld_piv := CRobT(\Tool:=tWeldGun\WObj:=wobjHsideplate);
        TPWrite "SRH29X XYZ:="\Pos:=SRH29X.trans;
		MoveL Offs(XH29E,80,0,0), v500, z1, tWeldGun\WObj:=wobjHpivot;
		Search_1D SRH0X\SearchStop:=X_Temp, Offs(XH0E,50,0,0), XH0E, v300, tWeldGun\WObj:=wobjHanchor\SchSpeed:=10;
		MoveL X_Temp, v50, fine, tWeldGun\WObj:=wobjHanchor;
        WaitTime\InPos, .1;
		Hx_weld_anchor := CRobT(\Tool:=tWeldGun\WObj:=wobjHsideplate);
        TPWrite "SRH0X XYZ:="\Pos:=SRH0X.trans;
		MoveL Offs(XH0E,120,0,0), v500, z1, tWeldGun\WObj:=wobjHanchor;
		MoveL Offs(XH19E,120,0,0), v500, z1, tWeldGun\WObj:=wobjHtip;
		Search_1D SRH19X\SearchStop:=X_Temp, Offs(XH19E,50,0,0), XH19E, v300, tWeldGun\WObj:=wobjHtip\SchSpeed:=10;
		MoveL X_Temp, v50, fine, tWeldGun\WObj:=wobjHtip;
        WaitTime\InPos, .1;
		Hx_weld_tip := CRobT(\Tool:=tWeldGun\WObj:=wobjHsideplate);
        TPWrite "SRH19X XYZ:="\Pos:=SRH19X.trans;
		MoveL Offs(XH19E,120,0,0), v500, z1, tWeldGun\WObj:=wobjHtip;
		MoveJ halfwayhome_H, vExtMax, z1, tWeldGun\WObj:=wobjHsideplate;
        BACK2H:
	ENDPROC

	PROC SEARCH_Mx()
		ActUnit STN1;
	    AccSet 75, 75;
        !!!!!!MOVING TO THE 3 X SEARCHES FOR M
        MoveJ halfwayhome_M, vExtMax, z1, tWeldGun\WObj:=wobjHsideplate;
		MoveJ Offs(XM69E,80,-550,-50), v500, z1, tWeldGun\WObj:=wobjHtip;
		MoveL Offs(XM69E,80,0,0), v500, z1, tWeldGun\WObj:=wobjHtip;
		Search_1D SRM69X\SearchStop:=X_Temp, Offs(XM69E,50,0,0), XM69E, v300, tWeldGun\WObj:=wobjHtip\SchSpeed:=10;
  		MoveL X_Temp, v50, fine, tWeldGun\WObj:=wobjHtip;
        WaitTime\InPos, 0.2;
		Mx_weld_tip := CRobT(\Tool:=tWeldGun\WObj:=wobjHsideplate);
        TPWrite "SRM69X XYZ:="\Pos:=SRM69X.trans;
		MoveL Offs(XM69E,80,0,0), v500, z1, tWeldGun\WObj:=wobjHtip;
		MoveL Offs(XM69E,80,-350,40), v500, z1, tWeldGun\WObj:=wobjHtip;
		MoveL Offs(XM61E,80,-350,-80), v500, z1, tWeldGun\WObj:=wobjHanchor;
		MoveL Offs(XM61E,80,0,0), v500, z1, tWeldGun\WObj:=wobjHanchor;
		Search_1D SRM61X\SearchStop:=X_Temp, Offs(XM61E,50,0,0), XM61E, v300, tWeldGun\WObj:=wobjHanchor\SchSpeed:=10;
  		MoveL X_Temp, v50, fine, tWeldGun\WObj:=wobjHanchor;
        WaitTime\InPos, 0.2;
		Mx_weld_anchor := CRobT(\Tool:=tWeldGun\WObj:=wobjHsideplate);
        TPWrite "SRM61X XYZ:="\Pos:=SRM61X.trans;
		MoveL Offs(XM61E,80,0,0), v500, z1, tWeldGun\WObj:=wobjHanchor;
		MoveL Offs(XM61E,80,-350,-80), v500, z1, tWeldGun\WObj:=wobjHanchor;
        MoveL Offs(XM49E,60,-300,0), vExtMax, fine, tWeldGun\WObj:=wobjHpivot;
        MoveL Offs(XM49E,60,0,0), vExtMax, fine, tWeldGun\WObj:=wobjHpivot;
		Search_1D SRM49X\SearchStop:=X_Temp, Offs(XM49E,50,0,0), XM49E, v300, tWeldGun\WObj:=wobjHpivot\SchSpeed:=10;
  		MoveL X_Temp, v50, fine, tWeldGun\WObj:=wobjHpivot;
        WaitTime\InPos, 0.2;
		Mx_weld_piv := CRobT(\Tool:=tWeldGun\WObj:=wobjHsideplate);
        TPWrite "SRM49X XYZ:="\Pos:=SRM49X.trans;
        MoveL Offs(XM49E,60,0,0), v500, z1, tWeldGun\WObj:=wobjHpivot;
        MoveJ Offs(XM49E,60,-400,0), vExtMax, fine, tWeldGun\WObj:=wobjHpivot;
 		MoveJ halfwayhome_M, vExtMax, z1, tWeldGun\WObj:=wobjHsideplate;
        BACK2M:
	ENDPROC

	PROC SEARCH_Lx()
		ActUnit STN1;
	    AccSet 75, 75;
        !!!!!!MOVING TO THE 3 X SEARCHES FOR L
        MoveL halfwayhome_L, vExtMax, z1, tWeldGun\WObj:=wobjHsideplate;
		MoveL Offs(XL69E,80,0,0), v500, z1, tWeldGun\WObj:=wobjHtip;
		Search_1D SRL69X\SearchStop:=X_Temp, Offs(XL69E,50,0,0), XL69E, v300, tWeldGun\WObj:=wobjHtip\SchSpeed:=10;
  		MoveL X_Temp, v50, fine, tWeldGun\WObj:=wobjHtip;
        WaitTime\InPos, 0.2;
		Lx_weld_tip := CRobT(\Tool:=tWeldGun\WObj:=wobjHsideplate);
        TPWrite "SRL69X XYZ:="\Pos:=SRL69X.trans;
		MoveL Offs(XL69E,80,0,0), v500, z1, tWeldGun\WObj:=wobjHtip;
		MoveL Offs(XL61E,80,0,0), v500, z1, tWeldGun\WObj:=wobjHanchor;
		Search_1D SRL61X\SearchStop:=X_Temp, Offs(XL61E,50,0,0), XL61E, v300, tWeldGun\WObj:=wobjHanchor\SchSpeed:=10;
  		MoveL X_Temp, v50, fine, tWeldGun\WObj:=wobjHanchor;
        WaitTime\InPos, 0.2;
		Lx_weld_anchor := CRobT(\Tool:=tWeldGun\WObj:=wobjHsideplate) ;
        TPWrite "SRL61X XYZ:="\Pos:=SRL61X.trans;
		MoveL Offs(XL61E,80,0,0), v500, z1, tWeldGun\WObj:=wobjHanchor;
		MoveL XL69air2, vExtMax, z1, tWeldGun\WObj:=wobjHsideplate;
		MoveJ XL4air23, vExtMax, z1, tWeldGun\WObj:=wobjHsideplate;
        MoveJ Offs(XL49E,120,0,50), vExtMax, fine, tWeldGun\WObj:=wobjHpivot;
        MoveL Offs(XL49E,80,0,0), vExtMax, fine, tWeldGun\WObj:=wobjHpivot;
		Search_1D SRL49X\SearchStop:=X_Temp, Offs(XL49E,50,0,0), XL49E, v300, tWeldGun\WObj:=wobjHpivot\SchSpeed:=10;
  		MoveL X_Temp, v50, fine, tWeldGun\WObj:=wobjHpivot;
        WaitTime\InPos, 0.2;
		Lx_weld_piv := CRobT(\Tool:=tWeldGun\WObj:=wobjHsideplate);
        TPWrite "SRL49X XYZ:="\Pos:=SRL49X.trans;
        MoveL Offs(XL49E,80,0,0), vExtMax, fine, tWeldGun\WObj:=wobjHpivot;
        MoveJ Offs(XL49E,100,0,50), vExtMax, fine, tWeldGun\WObj:=wobjHpivot;
        MoveJ XL4air23, vExtMax, z1, tWeldGun\WObj:=wobjHsideplate;
        MoveJ halfwayhome_L, vExtMax, z1, tWeldGun\WObj:=wobjHsideplate;
        BACK2L:
	ENDPROC

	PROC WELD_ONE()
		AccSet 50, 50;
		DROPSOME_ARM_DATA;
		CheckWNUMS;
        THIS_ARM_REVs;
        ZERO_X_A_ALL;
        ZERO_X_B_ALL;
        ZERO_X_G_ALL;
        ZERO_X_H_ALL;
        ZERO_X_L_ALL;
        ZERO_X_M_ALL;
        pure_adj18HTIP;
		WELDtip;
		TorchClean;
		WELD_THE_ANCHOR YY36, ZZ33;
		TorchClean;
		pausetoTACKFRONTWRAP;
		WELDpivot_18H;
		TorchClean;
		WELD_60s_ALL;
		TorchClean;
        WELD_41_42_46s;
		TorchClean;
		pausetoTACKBACKWRAP;
		WELDBACKWRAPtotip;
		TorchClean;
       IF pivCAM = TRUE THEN
        Weld_Piv0ut_2FWrap;
        TorchClean;
       ENDIF
        WELD_49_47_45s;
	    TorchClean;
	    WELD_30s_ALL;
	    TorchClean;
	    WELDFRONTWRAPpivotandtip;
	    TorchClean;
		WELD_20s_ALL;
		TorchClean;
		MoveToPark;
		COMPLETED;
	ENDPROC

	PROC WNUMB()
     !!!!!!! PUTS THE LOAD VARIABLES IN !!!!
     Load_6806128R4;
     ENDPROC

	PROC COMPLETED()
        TPWrite "  THIS PART IS COMPLETED!       ";
        TPWrite "  PLEASE REMOVE THE PART        ";
        TPWrite "  RELOAD AND BEGIN AGAIN        ";
	ENDPROC

	PROC W6806128rev4_PR3()
        WNUMB;
        WELD_ONE;
	ENDPROC

	PROC DROPSOME_ARM_DATA()
        WNUMB;
        WaitTime\InPos, .2;
        CheckWNUMS;
        WaitTime\InPos, .2;
        TIP_WOBJ wobjHtip, WTIPANGLE;
        WaitTime\InPos, .2;
        PIVOT_WOBJ wobjHpivot, WOTOX, WPIVOTANGLE, HFIXCONST;
        WaitTime\InPos, .2;
        ANCHOR_WOBJ wobjHanchor, WANCHORY, WANCHORz, WANCHORANGLE, HFIXCONST;
        WaitTime\InPos, .2;
        HSIDEPLATE_WOBJ wobjHsideplate, HFIXCONST;
        WaitTime\InPos, .2;
        ANCHOR_WOBJ wobjHanchor, WANCHORY, WANCHORz, WANCHORANGLE, HFIXCONST;
        WaitTime\InPos, .2;
        Pivot_Wobj_Cam wobj_PivCam, WPIVOTANGLE;
        WaitTime\InPos, .2;
        MoveToHome ;
        outta_here:
    ENDPROC

	PROC THIS_ARM_REVs()

        TPWrite "THE PART RUNNING IS  "\Num:=THISPROGRAM;
        TPWrite "THE PRINT REVISION IS  "\Num:=THISPARTREV;
        TPWrite "THE PROGRAM REVISION IS  "\Num:=THISPROGREV;

	ENDPROC

	PROC yTIP_WOBJ_DOCTOR(INOUT wobjdata wobjHtip,num WTIPANGLE)
        !!!!!!Created to adjust tip wobj by a search result!!!!!
        !!!!!! R-0 01-11-16 sy !!!!!!!!!!!!!!!
        !!!!!! R-1 01-20-16  sy !!!!!!!!!!!!!!!

        IF ADJTIPSRCH > 0 THEN
        	WTIPANGLEadj := WTIPANGLE - Abs(ADJTIPSRCH);
        ELSE
        	WTIPANGLEadj := WTIPANGLE + Abs(ADJTIPSRCH);
        ENDIF

		nZ := 0;
		nY := 0;
		nX := WTIPANGLEadj;
        wobjHtip := obSTN1;
        FRAME_TIP.rot := OrientZYX(nZ,nY,nX);
		FRAME_TIP.trans.x := 0 + FRAME_BASE.trans.x;
		FRAME_TIP.trans.y := -14 + FRAME_BASE.trans.y;
		FRAME_TIP.trans.z := 204.5 + FRAME_BASE.trans.z;
		wobjHtip.oframe := FRAME_TIP;
        WaitTime 0.5;
        TPWrite "ORIGINAL WTIPANGLE IS :="\num := WTIPANGLE;
        TPWrite ".............";
        TPWrite "WTIPANGLE ADJUSTED IS :="\num := WTIPANGLEadj;
        WaitTime 2;

    ENDPROC

	PROC pure_adj18HTIP()

        !!!!!!Created to work with yTIP_WOBJ_DOCTOR to adjust tip wobj by a search result!!!!!
        !!!!!! R-0 01-11-16 sy !!!!!!!!!!!!!!!
        TPErase;
        TPWrite "                                          ";
        TPWrite "                                          ";
        TPWrite "     THIS IS THE pure_adj18HTIP PROGRAM       ";
        TPWrite "                                          ";
        WaitTime 1;
     	AccSet 50, 50;
        WNUMB;
     	ActUnit STN1;
		MoveJ pjthomeSTA1zero, vCellSpeed, fine, tWeldGun\WObj:=wobj0;
		MoveJ Offs(SPT50E,-500,-50,100), vExtMax, z1, tWeldGun\WObj:=wobjHtip;
		PDispOff;
		TPErase;
		MoveL Offs(SPU650HRE,-120,60,0), vExtMax, z1, tWeldGun\WObj:=wobjHtip;
        !!!!!SRG11 is for the right side of the part at 0,0 degrees!!!!
		Search_1D SRG11, Offs(SPU650HRE,0,20,0), SPU650HRE, v200, tWeldGun\WObj:=wobjHtip\SchSpeed:=10;
        TPWrite "Y RIGHT SIDE of TIP is off zero by:="\Pos:=SRG11.trans;
		MoveL Offs(SPU650HRE,-120,60,0), vExtMax, z1, tWeldGun\WObj:=wobjHtip;
		MoveL Offs(SPT50E,-500,-50,100), vExtMax, z1, tWeldGun\WObj:=wobjHtip;
		MoveJ Offs(SPT40E,500,-50,100), vExtMax, z1, tWeldGun\WObj:=wobjHtip;
		MoveL Offs(SPU600HLE,120,60,0), vExtMax, z1, tWeldGun\WObj:=wobjHtip;
        !!!!!SRG12 is for the left side of the part at 0,0 degrees!!!!
		Search_1D SRG12, Offs(SPU600HLE,0,20,0), SPU600HLE, v200, tWeldGun\WObj:=wobjHtip\SchSpeed:=10;
       TPWrite "Y LEFT SIDE of TIP is off zero by:="\Pos:=SRG12.trans;
		MoveL Offs(SPU600HLE,120,60,0), v200, z1, tWeldGun\WObj:=wobjHtip;
        SRaveofG11G12.trans.y:= (SRG12.trans.y + SRG11.trans.y)/2;
        TPWrite "avg.search distance off true Y is:="\Pos:=SRaveofG11G12.trans;
        WaitTime 2;
        ADJTIPSRCH := ASin(SRaveofG11G12.trans.y/230);
        TPWrite "WTIPANGLE to be ADJUSTED by :="\num := ADJTIPSRCH;
        TPWrite "   DEGREES   ";
        WaitTime 2;
        !Stop;
		yTIP_WOBJ_DOCTOR wobjHtip, WTIPANGLE;
		MoveL Offs(SPT40E,500,-50,100), vExtMax, z1, tWeldGun\WObj:=wobjHtip;
		MoveJ pjthomeSTA1zero, vCellSpeed, fine, tWeldGun\WObj:=wobj0;
		FIXTIPDONE:
		bottom:
	ENDPROC

	PROC ZERO_X_A_ALL()
        A39.trans.x := 0;
        A38.trans.x := 0;
        A37.trans.x := 0;
        A36K.trans.x := 0;
        A36.trans.x := 0;
        A35.trans.x := 0;
        A33K.trans.x := 0;
        A33.trans.x := 0;
        A30.trans.x := 0;
        A31.trans.x := 0;
        A32.trans.x := 0;
        A325.trans.x := 0;
        A34.trans.x := 0;
	ENDPROC

	PROC ZERO_X_B_ALL()
        B39.trans.x := 0;
        B38.trans.x := 0;
        B37.trans.x := 0;
        B36K.trans.x := 0;
        B36.trans.x := 0;
        B35.trans.x := 0;
        B33K.trans.x := 0;
        B33.trans.x := 0;
        B30.trans.x := 0;
        B31.trans.x := 0;
        B32.trans.x := 0;
        B325.trans.x := 0;
        B34.trans.x := 0;
	ENDPROC

	PROC ZERO_X_G_ALL()
         G19.trans.x := 0;
         G18.trans.x := 0;
         G16.trans.x := 0;
         G15.trans.x := 0;
         G15K.trans.x := 0;
         G10.trans.x := 0;
         G21.trans.x := 0;
         G21K.trans.x := 0;
         G29.trans.x := 0;
         G27.trans.x := 0;
         G25.trans.x := 0;
         G23.trans.x := 0;
         G0.trans.x := 0;
 	ENDPROC

	PROC ZERO_X_H_ALL()
         H19.trans.x := 0;
         H18.trans.x := 0;
         H16.trans.x := 0;
         H15.trans.x := 0;
         H15K.trans.x := 0;
         H10.trans.x := 0;
         H21.trans.x := 0;
         H21K.trans.x := 0;
         H29.trans.x := 0;
         H27.trans.x := 0;
         H25.trans.x := 0;
         H23.trans.x := 0;
         H0.trans.x := 0;
 	ENDPROC

    PROC ZERO_X_L_ALL()
     L41.trans.x := 0;
     L40.trans.x := 0;
     L42.trans.x := 0;
     L43.trans.x := 0;
     L44.trans.x := 0;
     L45.trans.x := 0;
     L46.trans.x := 0;
     L47.trans.x := 0;
     L48.trans.x := 0;
     L49.trans.x := 0;
     L50.trans.x := 0;
     L60.trans.x := 0;
     L61.trans.x := 0;
     L62.trans.x := 0;
     L63.trans.x := 0;
     L64.trans.x := 0;
     L65.trans.x := 0;
     L66.trans.x := 0;
     L67.trans.x := 0;
     L64K.trans.x := 0;
     L65K.trans.x := 0;
     L66K.trans.x := 0;
     L67K.trans.x := 0;
     L68.trans.x := 0;
     L69.trans.x := 0;
     L70.trans.x := 0;
    ENDPROC

   	PROC ZERO_X_M_ALL()
    M40.trans.x := 0;
    M41.trans.x := 0;
    M42.trans.x := 0;
    M43.trans.x := 0;
    M44.trans.x := 0;
    M45.trans.x := 0;
    M46.trans.x := 0;
    M47.trans.x := 0;
    M48.trans.x := 0;
    M49.trans.x := 0;
    M50.trans.x := 0;
    M60.trans.x := 0;
    M61.trans.x := 0;
    M62.trans.x := 0;
    M63.trans.x := 0;
    M64.trans.x := 0;
    M65.trans.x := 0;
    M66.trans.x := 0;
    M67.trans.x := 0;
    M64K.trans.x := 0;
    M65K.trans.x := 0;
    M66K.trans.x := 0;
    M67K.trans.x := 0;
    M68.trans.x := 0;
    M69.trans.x := 0;
    M70.trans.x := 0;
    ENDPROC

    PROC SET_G20s_X()
        G_X_POINT_SETTER  G19;
        G_X_POINT_SETTER  G18;
        G_X_POINT_SETTER  G16;
        G_X_POINT_SETTER  G15;
        G_X_POINT_SETTER  G15K;
        G_X_POINT_SETTER  G10;
        G_X_POINT_SETTER  G21K;
        G_X_POINT_SETTER  G21;
        G_X_POINT_SETTER  G0;

        G_X_POINT_SETTER  G23;
        G_X_POINT_SETTER  G24;
        G_X_POINT_SETTER  G25;
        G_X_POINT_SETTER  G26;
        G_X_POINT_SETTER  G27;
        G_X_POINT_SETTER  G28;
        G_X_POINT_SETTER  G29;
     aplace:
    ENDPROC

    PROC SET_H20s_X()
        H_X_POINT_SETTER  H19;
        H_X_POINT_SETTER  H18;
        H_X_POINT_SETTER  H16;
        H_X_POINT_SETTER  H15;
        H_X_POINT_SETTER  H15K;
        H_X_POINT_SETTER  H10;
        H_X_POINT_SETTER  H21K;
        H_X_POINT_SETTER  H21;
        H_X_POINT_SETTER  H0;

        H_X_POINT_SETTER  H23;
        H_X_POINT_SETTER  H24;
        H_X_POINT_SETTER  H25;
        H_X_POINT_SETTER  H26;
        H_X_POINT_SETTER  H28;
        H_X_POINT_SETTER  H27;
        H_X_POINT_SETTER  H29;
     aplace:
    ENDPROC

    PROC SET_A30s_X()
        A_X_POINT_SETTER  A39;
        A_X_POINT_SETTER  A38;
        A_X_POINT_SETTER  A37;
        A_X_POINT_SETTER  A36;
        A_X_POINT_SETTER  A36K;
        A_X_POINT_SETTER  A35;
        A_X_POINT_SETTER  A34;
        A_X_POINT_SETTER  A33;
        A_X_POINT_SETTER  A33K;
        A_X_POINT_SETTER  A32;
        A_X_POINT_SETTER  A325;
        A_X_POINT_SETTER  A31;
        A_X_POINT_SETTER  A30;
      aplace:
    ENDPROC

    PROC SET_B30s_X()
        B_X_POINT_SETTER  B39;
        B_X_POINT_SETTER  B38;
        B_X_POINT_SETTER  B37;
        B_X_POINT_SETTER  B36;
        B_X_POINT_SETTER  B36K;
        B_X_POINT_SETTER  B35;
        B_X_POINT_SETTER  B34;
        B_X_POINT_SETTER  B33;
        B_X_POINT_SETTER  B33K;
        B_X_POINT_SETTER  B32;
        B_X_POINT_SETTER  B325;
        B_X_POINT_SETTER  B31;
        B_X_POINT_SETTER  B30;
       aplace:
    ENDPROC

    PROC SET_M40s_X()
        M_X_POINT_SETTER  M41;
        M_X_POINT_SETTER  M42;
        M_X_POINT_SETTER  M43;
        M_X_POINT_SETTER  M44;
        M_X_POINT_SETTER  M45;
        M_X_POINT_SETTER  M46;
        M_X_POINT_SETTER  M47;
        M_X_POINT_SETTER  M48;
        M_X_POINT_SETTER  M49;
       TAG_A_LONG_LM50 M50, AA49, M49, 15;
       aplace:
    ENDPROC

    PROC SET_L40s_X()
        L_X_POINT_SETTER  L41;
        L_X_POINT_SETTER  L42;
        L_X_POINT_SETTER  L43;
        L_X_POINT_SETTER  L44;
        L_X_POINT_SETTER  L45;
        L_X_POINT_SETTER  L46;
        L_X_POINT_SETTER  L47;
        L_X_POINT_SETTER  L48;
        L_X_POINT_SETTER  L49;
      TAG_A_LONG_LM50 L50, AA49, L49, 15;
      aplace:
    ENDPROC

    PROC SET_L60s_X()
        L_X_POINT_SETTER  L69;
        L_X_POINT_SETTER  L68;
        L_X_POINT_SETTER  L67K;
        L_X_POINT_SETTER  L67;
        L_X_POINT_SETTER  L66K;
        L_X_POINT_SETTER  L66;
        L_X_POINT_SETTER  L65K;
        L_X_POINT_SETTER  L65;
        L_X_POINT_SETTER  L64K;
        L_X_POINT_SETTER  L64;
        L_X_POINT_SETTER  L63;
        L_X_POINT_SETTER  L62;
        L_X_POINT_SETTER  L61;
        TAG_A_LONG_LM70 L70, AA69, L69, 15;
    aplace:
    ENDPROC

    PROC SET_M60s_X()
        M_X_POINT_SETTER M69;
        M_X_POINT_SETTER M68;
        M_X_POINT_SETTER M67K;
        M_X_POINT_SETTER M67;
        M_X_POINT_SETTER M66K;
        M_X_POINT_SETTER M66;
        M_X_POINT_SETTER M65K;
        M_X_POINT_SETTER M65;
        M_X_POINT_SETTER M64K;
        M_X_POINT_SETTER M64;
        M_X_POINT_SETTER M63;
        M_X_POINT_SETTER M62;
        M_X_POINT_SETTER M61;
        TAG_A_LONG_LM70 M70, AA69, M69, 15;
       aplace:
    ENDPROC

!!!!!!!!!!!!!!!!!!!!!!!!!!!!!!!!!!!!!!!!!!!!!!!!!!!!!!!!!!!!
!!!!!!!!!!!!!!!!!!!!!!!!!!!!!!!!!!!!!!!!!!!!!!!!!!!!!!!!!!!!
    PROC PivGXPJ_Cam_18_R1(INOUT
           ROBTARGET G_PJ_XCAM)

        SP_GPivCam_PJ_Ye.trans.X := G_PJ_XCAM.TRANS.X + NOZZLE_RADIUS + 8;
        SP_GPivCam_PJ_Ys.trans.X := G_PJ_XCAM.TRANS.X + NOZZLE_RADIUS + 8;

        SP_GPivCAM_PJ_Ze.trans.X := G_PJ_XCAM.TRANS.X + NOZZLE_RADIUS + 8;
        SP_GPivCAM_PJ_Zs.trans.X := G_PJ_XCAM.TRANS.X + NOZZLE_RADIUS + 8;

        G_PJCam_1st_s.TRANS.X  :=  G_PJ_XCAM.TRANS.X + NOZZLE_RADIUS - STICK_OUT ;
        G_PJCam_1st_sm.TRANS.X :=  G_PJ_XCAM.TRANS.X + NOZZLE_RADIUS - STICK_OUT ;
        G_PJCam_1st_em.TRANS.X :=  G_PJ_XCAM.TRANS.X + NOZZLE_RADIUS - STICK_OUT ;
        G_PJCam_1st_e.TRANS.X  :=  G_PJ_XCAM.TRANS.X + NOZZLE_RADIUS - STICK_OUT ;

        G_PJCam_2ND_s.TRANS.X  :=  G_PJ_XCAM.TRANS.X + NOZZLE_RADIUS - STICK_OUT ;
        G_PJCam_2ND_sm.TRANS.X :=  G_PJ_XCAM.TRANS.X + NOZZLE_RADIUS - STICK_OUT ;
        G_PJCam_2ND_em.TRANS.X :=  G_PJ_XCAM.TRANS.X + NOZZLE_RADIUS - STICK_OUT ;
        G_PJCam_2ND_e.TRANS.X  :=  G_PJ_XCAM.TRANS.X + NOZZLE_RADIUS - STICK_OUT ;

        G_PJCam_3RD_s.TRANS.X  :=  G_PJ_XCAM.TRANS.X + NOZZLE_RADIUS - STICK_OUT ;
        G_PJCam_3RD_sm.TRANS.X :=  G_PJ_XCAM.TRANS.X + NOZZLE_RADIUS - STICK_OUT ;
        G_PJCam_3RD_em.TRANS.X :=  G_PJ_XCAM.TRANS.X + NOZZLE_RADIUS - STICK_OUT ;
        G_PJCam_3RD_e.TRANS.X  :=  G_PJ_XCAM.TRANS.X + NOZZLE_RADIUS - STICK_OUT ;

        G_PJCam_4TH_s.TRANS.X  :=  G_PJ_XCAM.TRANS.X + NOZZLE_RADIUS - STICK_OUT ;
        G_PJCam_4TH_sm.TRANS.X :=  G_PJ_XCAM.TRANS.X + NOZZLE_RADIUS - STICK_OUT ;
        G_PJCam_4TH_em.TRANS.X :=  G_PJ_XCAM.TRANS.X + NOZZLE_RADIUS - STICK_OUT ;
        G_PJCam_4TH_e.TRANS.X  :=  G_PJ_XCAM.TRANS.X + NOZZLE_RADIUS - STICK_OUT ;

        G_PJCam_5TH_s.TRANS.X  :=  G_PJ_XCAM.TRANS.X + NOZZLE_RADIUS - STICK_OUT ;
        G_PJCam_5TH_sm.TRANS.X :=  G_PJ_XCAM.TRANS.X + NOZZLE_RADIUS - STICK_OUT ;
        G_PJCam_5TH_em.TRANS.X :=  G_PJ_XCAM.TRANS.X + NOZZLE_RADIUS - STICK_OUT ;
        G_PJCam_5TH_e.TRANS.X  :=  G_PJ_XCAM.TRANS.X + NOZZLE_RADIUS - STICK_OUT ;


        SP_GCAM_PjEDGE_S.trans.x := G_PJ_XCAM.TRANS.X + NOZZLE_RADIUS;
        SP_GCAM_PjEDGE_E.trans.x := G_PJ_XCAM.TRANS.X + NOZZLE_RADIUS;
        SP_GCAM_PjJOINT_S.trans.x := G_PJ_XCAM.TRANS.X + NOZZLE_RADIUS;
        SP_GCAM_PjJOINT_E.trans.x := G_PJ_XCAM.TRANS.X + NOZZLE_RADIUS;

       GX_PJ_DUNN:
    ENDPROC

    PROC PivHXPJ_Cam_18_R1(INOUT
           ROBTARGET H_PJ_XCAM)

        SP_HPivCam_PJ_Ye.trans.X :=  H_PJ_XCAM.TRANS      .X - NOZZLE_RADIUS -8 ;
        SP_HPivCam_PJ_Ys.trans.X :=  H_PJ_XCAM.TRANS      .X - NOZZLE_RADIUS -8 ;

        SP_HPivCam_PJ_Ze.trans.X :=  H_PJ_XCAM.TRANS      .X - NOZZLE_RADIUS -8 ;
        SP_HPivCam_PJ_Zs.trans.X :=  H_PJ_XCAM.TRANS      .X - NOZZLE_RADIUS -8 ;

        H_PJCam_1st_s.TRANS.X  :=  H_PJ_XCAM.TRANS.X - NOZZLE_RADIUS + STICK_OUT  ;
        H_PJCam_1st_sm.TRANS.X :=  H_PJ_XCAM.TRANS.X - NOZZLE_RADIUS + STICK_OUT  ;
        H_PJCam_1st_em.TRANS.X :=  H_PJ_XCAM.TRANS.X - NOZZLE_RADIUS + STICK_OUT  ;
        H_PJCam_1st_e.TRANS.X  :=  H_PJ_XCAM.TRANS.X - NOZZLE_RADIUS + STICK_OUT  ;

        H_PJCam_2ND_s.TRANS.X  :=  H_PJ_XCAM.TRANS.X - NOZZLE_RADIUS + STICK_OUT  ;
        H_PJCam_2ND_sm.TRANS.X :=  H_PJ_XCAM.TRANS.X - NOZZLE_RADIUS + STICK_OUT  ;
        H_PJCam_2ND_em.TRANS.X :=  H_PJ_XCAM.TRANS.X - NOZZLE_RADIUS + STICK_OUT  ;
        H_PJCam_2ND_e.TRANS.X  :=  H_PJ_XCAM.TRANS.X - NOZZLE_RADIUS + STICK_OUT  ;

        H_PJCam_3RD_s.TRANS.X  :=  H_PJ_XCAM.TRANS.X - NOZZLE_RADIUS + STICK_OUT  ;
        H_PJCam_3RD_sm.TRANS.X :=  H_PJ_XCAM.TRANS.X - NOZZLE_RADIUS + STICK_OUT  ;
        H_PJCam_3RD_em.TRANS.X :=  H_PJ_XCAM.TRANS.X - NOZZLE_RADIUS + STICK_OUT  ;
        H_PJCam_3RD_e.TRANS.X  :=  H_PJ_XCAM.TRANS.X - NOZZLE_RADIUS + STICK_OUT  ;

        H_PJCam_4TH_s.TRANS.X  :=  H_PJ_XCAM.TRANS.X - NOZZLE_RADIUS + STICK_OUT  ;
        H_PJCam_4TH_sm.TRANS.X :=  H_PJ_XCAM.TRANS.X - NOZZLE_RADIUS + STICK_OUT  ;
        H_PJCam_4TH_em.TRANS.X :=  H_PJ_XCAM.TRANS.X - NOZZLE_RADIUS + STICK_OUT  ;
        H_PJCam_4TH_e.TRANS.X  :=  H_PJ_XCAM.TRANS.X - NOZZLE_RADIUS + STICK_OUT  ;

        H_PJCam_5TH_s.TRANS.X  :=  H_PJ_XCAM.TRANS.X - NOZZLE_RADIUS + STICK_OUT  ;
        H_PJCam_5TH_sm.TRANS.X :=  H_PJ_XCAM.TRANS.X - NOZZLE_RADIUS + STICK_OUT  ;
        H_PJCam_5TH_em.TRANS.X :=  H_PJ_XCAM.TRANS.X - NOZZLE_RADIUS + STICK_OUT  ;
        H_PJCam_5TH_e.TRANS.X  :=  H_PJ_XCAM.TRANS.X - NOZZLE_RADIUS + STICK_OUT  ;

        SP_HCAM_PJEDGE_S.TRANS.X  :=  H_PJ_XCAM.TRANS.X - NOZZLE_RADIUS  ;
        SP_HCAM_PJEDGE_E.TRANS.X  :=  H_PJ_XCAM.TRANS.X - NOZZLE_RADIUS  ;
        SP_HCAM_PJJOINT_S.TRANS.X  :=  H_PJ_XCAM.TRANS.X - NOZZLE_RADIUS  ;
        SP_HCAM_PJJOINT_E.TRANS.X  :=  H_PJ_XCAM.TRANS.X - NOZZLE_RADIUS  ;
       GX_PJ_DUNN:
    ENDPROC

    PROC PivGXPJ_Rnd(INOUT
          ROBTARGET G_PJ_XRND)

        SP_GPivRnd_PJ_Ye.trans.X := G_PJ_XRND.TRANS.X - NOZZLE_RADIUS - SIDEPLATE ;
        SP_GPivRnd_PJ_Ys.trans.X := G_PJ_XRND.TRANS.X - NOZZLE_RADIUS - SIDEPLATE ;

        SP_GPivRND_PJ_Ze.trans.X := G_PJ_XRND.TRANS.X - NOZZLE_RADIUS - SIDEPLATE ;
        SP_GPivRND_PJ_Zs.trans.X := G_PJ_XRND.TRANS.X - NOZZLE_RADIUS - SIDEPLATE ;

        G_PJRnd_1st_s.TRANS.X  :=  G_PJ_XRND.TRANS.X - NOZZLE_RADIUS;
        G_PJRnd_1st_sm.TRANS.X :=  G_PJ_XRND.TRANS.X - NOZZLE_RADIUS ;
        G_PJRnd_1st_em.TRANS.X :=  G_PJ_XRND.TRANS.X - NOZZLE_RADIUS ;
        G_PJRnd_1st_e.TRANS.X  :=  G_PJ_XRND.TRANS.X - NOZZLE_RADIUS ;

        G_PJRnd_2ND_s.TRANS.X  :=  G_PJ_XRND.TRANS.X - NOZZLE_RADIUS ;
        G_PJRnd_2ND_sm.TRANS.X :=  G_PJ_XRND.TRANS.X - NOZZLE_RADIUS ;
        G_PJRnd_2ND_em.TRANS.X :=  G_PJ_XRND.TRANS.X - NOZZLE_RADIUS ;
        G_PJRnd_2ND_e.TRANS.X  :=  G_PJ_XRND.TRANS.X - NOZZLE_RADIUS ;

        G_PJRnd_3RD_s.TRANS.X  :=  G_PJ_XRND.TRANS.X - NOZZLE_RADIUS ;
        G_PJRnd_3RD_sm.TRANS.X :=  G_PJ_XRND.TRANS.X - NOZZLE_RADIUS ;
        G_PJRnd_3RD_em.TRANS.X :=  G_PJ_XRND.TRANS.X - NOZZLE_RADIUS ;
        G_PJRnd_3RD_e.TRANS.X  :=  G_PJ_XRND.TRANS.X - NOZZLE_RADIUS ;

        G_PJRnd_4TH_s.TRANS.X  :=  G_PJ_XRND.TRANS.X - NOZZLE_RADIUS ;
        G_PJRnd_4TH_sm.TRANS.X :=  G_PJ_XRND.TRANS.X - NOZZLE_RADIUS ;
        G_PJRnd_4TH_em.TRANS.X :=  G_PJ_XRND.TRANS.X - NOZZLE_RADIUS ;
        G_PJRnd_4TH_e.TRANS.X  :=  G_PJ_XRND.TRANS.X - NOZZLE_RADIUS ;

        SP_GRnd_PJEDGE_S.TRANS.X :=  G_PJ_XRND.TRANS.X - NOZZLE_RADIUS  ;
        SP_GRnd_PJEDGE_E.TRANS.X :=  G_PJ_XRND.TRANS.X - NOZZLE_RADIUS  ;

        SP_GRnd_PJJOINT_S.TRANS.X :=  G_PJ_XRND.TRANS.X - NOZZLE_RADIUS  ;
        SP_GRnd_PJJOINT_E.TRANS.X :=  G_PJ_XRND.TRANS.X - NOZZLE_RADIUS  ;

       GX_PJ_DUNN:
    ENDPROC

    PROC PivHXPJ_Rnd(INOUT
           ROBTARGET H_PJ_XRND)

        SP_HPivRnd_PJ_Ye.trans.X :=  H_PJ_XRND.TRANS.X + NOZZLE_RADIUS + SIDEPLATE ;
        SP_HPivRnd_PJ_Ys.trans.X :=  H_PJ_XRND.TRANS.X + NOZZLE_RADIUS + SIDEPLATE ;

        SP_HPivRnd_PJ_Ze.trans.X :=  H_PJ_XRND.TRANS.X + NOZZLE_RADIUS + SIDEPLATE;
        SP_HPivRnd_PJ_Zs.trans.X :=  H_PJ_XRND.TRANS.X + NOZZLE_RADIUS + SIDEPLATE;

        H_PJRnd_1st_s.TRANS.X  :=  H_PJ_XRND.TRANS.X + NOZZLE_RADIUS;
        H_PJRnd_1st_sm.TRANS.X :=  H_PJ_XRND.TRANS.X + NOZZLE_RADIUS ;
        H_PJRnd_1st_em.TRANS.X :=  H_PJ_XRND.TRANS.X + NOZZLE_RADIUS ;
        H_PJRnd_1st_e.TRANS.X  :=  H_PJ_XRND.TRANS.X + NOZZLE_RADIUS  ;

        H_PJRnd_2ND_s.TRANS.X  :=  H_PJ_XRND.TRANS.X + NOZZLE_RADIUS ;
        H_PJRnd_2ND_sm.TRANS.X :=  H_PJ_XRND.TRANS.X + NOZZLE_RADIUS ;
        H_PJRnd_2ND_em.TRANS.X :=  H_PJ_XRND.TRANS.X + NOZZLE_RADIUS ;
        H_PJRnd_2ND_e.TRANS.X  :=  H_PJ_XRND.TRANS.X + NOZZLE_RADIUS ;

        H_PJRnd_3RD_s.TRANS.X  :=  H_PJ_XRND.TRANS.X + NOZZLE_RADIUS ;
        H_PJRnd_3RD_sm.TRANS.X :=  H_PJ_XRND.TRANS.X + NOZZLE_RADIUS ;
        H_PJRnd_3RD_em.TRANS.X :=  H_PJ_XRND.TRANS.X + NOZZLE_RADIUS ;
        H_PJRnd_3RD_e.TRANS.X  :=  H_PJ_XRND.TRANS.X + NOZZLE_RADIUS ;

        H_PJRnd_4TH_s.TRANS.X  :=  H_PJ_XRND.TRANS.X + NOZZLE_RADIUS - STICK_OUT ;
        H_PJRnd_4TH_sm.TRANS.X :=  H_PJ_XRND.TRANS.X + NOZZLE_RADIUS - STICK_OUT ;
        H_PJRnd_4TH_em.TRANS.X :=  H_PJ_XRND.TRANS.X + NOZZLE_RADIUS - STICK_OUT ;
        H_PJRnd_4TH_e.TRANS.X  :=  H_PJ_XRND.TRANS.X + NOZZLE_RADIUS - (1.5 * STICK_OUT) ;

        SP_HRnd_PJEDGE_S.TRANS.X :=  H_PJ_XRND.TRANS.X + NOZZLE_RADIUS  ;
        SP_HRnd_PJEDGE_E.TRANS.X :=  H_PJ_XRND.TRANS.X + NOZZLE_RADIUS  ;

        SP_HRnd_PJJOINT_S.TRANS.X :=  H_PJ_XRND.TRANS.X + NOZZLE_RADIUS  ;
        SP_HRnd_PJJOINT_E.TRANS.X :=  H_PJ_XRND.TRANS.X + NOZZLE_RADIUS  ;
        WaitTime\InPos, 1;

        HX_PJ_DUNN:
    ENDPROC

    PROC PivGX18_Cam_18_R1(INOUT
        ROBTARGET G18_XCAM)

        SP_GPivCam_18_Ye.trans.X := G18_XCAM.TRANS.X - NOZZLE_RADIUS - SIDEPLATE +8 ;
        SP_GPivCam_18_Ys.trans.X := G18_XCAM.TRANS.X - NOZZLE_RADIUS - SIDEPLATE+8 ;

        SP_GPivCAM_18_Ze.trans.X := G18_XCAM.TRANS.X - NOZZLE_RADIUS - SIDEPLATE+8 ;
        SP_GPivCAM_18_Zs.trans.X := G18_XCAM.TRANS.X - NOZZLE_RADIUS - SIDEPLATE+8 ;

        G_CAM_1.TRANS.X := G18_XCAM.TRANS.X - NOZZLE_RADIUS + STICK_OUT ;
        G_CAM_2.TRANS.X := G18_XCAM.TRANS.X - NOZZLE_RADIUS + STICK_OUT ;
        G_CAM_3.TRANS.X := G18_XCAM.TRANS.X - NOZZLE_RADIUS + STICK_OUT ;
        G_CAM_4.TRANS.X := G18_XCAM.TRANS.X - NOZZLE_RADIUS + STICK_OUT ;
        G_CAM_5.TRANS.X := G18_XCAM.TRANS.X - NOZZLE_RADIUS + STICK_OUT ;
        G_CAM_6.TRANS.X := G18_XCAM.TRANS.X - NOZZLE_RADIUS + STICK_OUT ;
        G_CAM_7.TRANS.X := G18_XCAM.TRANS.X - NOZZLE_RADIUS + STICK_OUT ;
        G_CAM_8.TRANS.X := G18_XCAM.TRANS.X - NOZZLE_RADIUS + STICK_OUT ;

           gx18_dunn:
    ENDPROC

    PROC PivHX18_Cam_18_R1(INOUT
          ROBTARGET H18_XCAM)
           SP_HPivCam_18_Ye.trans.X :=  H18_XCAM.TRANS.X - NOZZLE_RADIUS - SIDEPLATE +8 ;
           SP_HPivCam_18_Ys.trans.X :=  H18_XCAM.TRANS.X - NOZZLE_RADIUS - SIDEPLATE +8 ;

           SP_HPivCam_18_Ze.trans.X :=  H18_XCAM.TRANS.X - NOZZLE_RADIUS - SIDEPLATE +8;
           SP_HPivCam_18_Zs.trans.X :=  H18_XCAM.TRANS.X - NOZZLE_RADIUS - SIDEPLATE +8;

           H_CAM_1.TRANS.X := H18_XCAM.TRANS.X - NOZZLE_RADIUS - STICK_OUT - SIDEPLATE ;
           H_CAM_2.TRANS.X := H18_XCAM.TRANS.X - NOZZLE_RADIUS - STICK_OUT - SIDEPLATE ;
           H_CAM_3.TRANS.X := H18_XCAM.TRANS.X - NOZZLE_RADIUS - STICK_OUT - SIDEPLATE ;
           H_CAM_4.TRANS.X := H18_XCAM.TRANS.X - NOZZLE_RADIUS - STICK_OUT - SIDEPLATE ;
           H_CAM_5.TRANS.X := H18_XCAM.TRANS.X - NOZZLE_RADIUS - STICK_OUT - SIDEPLATE ;
           H_CAM_6.TRANS.X := H18_XCAM.TRANS.X - NOZZLE_RADIUS - STICK_OUT - SIDEPLATE ;
           H_CAM_7.TRANS.X := H18_XCAM.TRANS.X - NOZZLE_RADIUS - STICK_OUT - SIDEPLATE ;
           H_CAM_8.TRANS.X := H18_XCAM.TRANS.X - NOZZLE_RADIUS - STICK_OUT - SIDEPLATE ;

           hx18_dunn:
    ENDPROC

    PROC PivGX18_Rnd(INOUT
             ROBTARGET G18_XRND)

           SP_GPivRnd_18_Ye.trans.X := G18_XRND.TRANS.X + NOZZLE_RADIUS ;
           SP_GPivRnd_18_Ys.trans.X := G18_XRND.TRANS.X + NOZZLE_RADIUS ;

           SP_GPivRND_18_Ze.trans.X := G18_XRND.TRANS.X + NOZZLE_RADIUS ;
           SP_GPivRND_18_Zs.trans.X := G18_XRND.TRANS.X + NOZZLE_RADIUS ;

           G_RND_1.TRANS.X := G18_XRND.TRANS.X + NOZZLE_RADIUS - STICK_OUT ;
           G_RND_2.TRANS.X := G18_XRND.TRANS.X + NOZZLE_RADIUS - STICK_OUT ;
           G_RND_3.TRANS.X := G18_XRND.TRANS.X + NOZZLE_RADIUS - STICK_OUT ;
           G_RND_4.TRANS.X := G18_XRND.TRANS.X + NOZZLE_RADIUS - STICK_OUT ;
           G_RND_5.TRANS.X := G18_XRND.TRANS.X + NOZZLE_RADIUS - STICK_OUT ;
           G_RND_6.TRANS.X := G18_XRND.TRANS.X + NOZZLE_RADIUS - STICK_OUT ;
           G_RND_7.TRANS.X := G18_XRND.TRANS.X + NOZZLE_RADIUS - STICK_OUT ;

           gx18_dunn:
    ENDPROC

    PROC PivHX18_Rnd(INOUT
               ROBTARGET H18_XRND)

           SP_HPivRnd_18_Ye.trans.X :=  H18_XRND.TRANS.X - NOZZLE_RADIUS ;
           SP_HPivRnd_18_Ys.trans.X :=  H18_XRND.TRANS.X - NOZZLE_RADIUS ;

           SP_HPivRnd_18_Ze.trans.X :=  H18_XRND.TRANS.X - NOZZLE_RADIUS ;
           SP_HPivRnd_18_Zs.trans.X :=  H18_XRND.TRANS.X - NOZZLE_RADIUS;

          H_RND_1.TRANS.X := H18_XRND.TRANS.X - NOZZLE_RADIUS + STICK_OUT ;
          H_RND_2.TRANS.X := H18_XRND.TRANS.X - NOZZLE_RADIUS + STICK_OUT ;
          H_RND_3.TRANS.X := H18_XRND.TRANS.X - NOZZLE_RADIUS + STICK_OUT ;
          H_RND_4.TRANS.X := H18_XRND.TRANS.X - NOZZLE_RADIUS + STICK_OUT ;
          H_RND_5.TRANS.X := H18_XRND.TRANS.X - NOZZLE_RADIUS + STICK_OUT ;
          H_RND_6.TRANS.X := H18_XRND.TRANS.X - NOZZLE_RADIUS + STICK_OUT ;
          H_RND_7.TRANS.X := H18_XRND.TRANS.X - NOZZLE_RADIUS + STICK_OUT ;
           Hx18_dunn:
    ENDPROC

    PROC PivG_SideYZ_XSET_18_R1(inout
            robtarget That_SIDE)

	SP_GRnd_Side_YS.TRANS.X :=  That_SIDE.TRANS.X + NOZZLE_RADIUS ;
	SP_GRnd_Side_YE.TRANS.X :=  That_SIDE.TRANS.X + NOZZLE_RADIUS ;
	SP_GRnd_Side_ZS.TRANS.X :=  That_SIDE.TRANS.X + NOZZLE_RADIUS ;
	SP_GRnd_Side_ZE.TRANS.X :=  That_SIDE.TRANS.X + NOZZLE_RADIUS ;

	SP_GCam_Side_YS.TRANS.X :=  That_SIDE.TRANS.X + NOZZLE_RADIUS +7 ;
	SP_GCam_Side_YE.TRANS.X :=  That_SIDE.TRANS.X + NOZZLE_RADIUS +7 ;
	SP_GCam_Side_ZS.TRANS.X :=  That_SIDE.TRANS.X + NOZZLE_RADIUS +7 ;
	SP_GCam_Side_ZE.TRANS.X :=  That_SIDE.TRANS.X + NOZZLE_RADIUS +7 ;

   !!!!!!!!!!!!!!!!!!!!!!!!!!!!!!!!!!!!!!!!!!!!!!!!!!!!!!!!!!!!!!!!!!!!!!!!!!!!!!!!!!!!
    GRnd_SidePIV_S.TRANS.X := That_SIDE.TRANS.X   ;
    GRnd_SidePIV_SM.TRANS.X := That_SIDE.TRANS.X  ;
    GRnd_SidePIV_M.TRANS.X := That_SIDE.TRANS.X   ;
    GRnd_SidePIV_EM.TRANS.X := That_SIDE.TRANS.X  ;
    GRnd_SidePIV_E.TRANS.X := That_SIDE.TRANS.X   ;

    GCam_SidePIV_S.TRANS.X := That_SIDE.TRANS.X + NOZZLE_RADIUS - STICK_OUT ;
    GCam_SidePIV_SM.TRANS.X := That_SIDE.TRANS.X + NOZZLE_RADIUS - STICK_OUT ;
    GCam_SidePIV_M.TRANS.X := That_SIDE.TRANS.X + NOZZLE_RADIUS - STICK_OUT ;
    GCam_SidePIV_EM.TRANS.X := That_SIDE.TRANS.X + NOZZLE_RADIUS - STICK_OUT;
    GCam_SidePIV_E.TRANS.X := That_SIDE.TRANS.X + NOZZLE_RADIUS - STICK_OUT ;
    !!!!!!!!!END!!!!!!!!!!
    ENDPROC

	PROC PivH_SideYZ_XSET_18_R1(inout
        robtarget This_SIDE)

	SP_HRnd_Side_YS.TRANS.X :=  This_SIDE.TRANS.X - NOZZLE_RADIUS ;
	SP_HRnd_Side_YE.TRANS.X :=  This_SIDE.TRANS.X - NOZZLE_RADIUS ;
	SP_HRnd_Side_ZS.TRANS.X :=  This_SIDE.TRANS.X - NOZZLE_RADIUS ;
	SP_HRnd_Side_ZE.TRANS.X :=  This_SIDE.TRANS.X - NOZZLE_RADIUS ;

	SP_HCam_Side_YS.TRANS.X :=  This_SIDE.TRANS.X - NOZZLE_RADIUS -7 ;
	SP_HCam_Side_YE.TRANS.X :=  This_SIDE.TRANS.X - NOZZLE_RADIUS -7 ;
	SP_HCam_Side_ZS.TRANS.X :=  This_SIDE.TRANS.X - NOZZLE_RADIUS -7 ;
	SP_HCam_Side_ZE.TRANS.X :=  This_SIDE.TRANS.X - NOZZLE_RADIUS -7 ;

    HCam_SidePIV_S.TRANS.X := This_SIDE.TRANS.X - nozzle_radius + stick_out;
    HCam_SidePIV_SM.TRANS.X := This_SIDE.TRANS.X - nozzle_radius + stick_out;
    HCam_SidePIV_M.TRANS.X := This_SIDE.TRANS.X - nozzle_radius + stick_out;
    HCam_SidePIV_EM.TRANS.X := This_SIDE.TRANS.X - nozzle_radius + stick_out;
    HCam_SidePIV_E.TRANS.X := This_SIDE.TRANS.X - nozzle_radius + stick_out;

    !!!!!!!!!!!!!!!!!!!!!!!!!!!!!!!!!!!!!!!!!!!!!!!!!!!!!!!!!!!!!!!!!!!!!!!!!!!!!!!!!!!!!
    HRnd_SidePIV_S.TRANS.X := This_SIDE.TRANS.X   ;
    HRnd_SidePIV_SM.TRANS.X := This_SIDE.TRANS.X  ;
    HRnd_SidePIV_M.TRANS.X := This_SIDE.TRANS.X   ;
    HRnd_SidePIV_EM.TRANS.X := This_SIDE.TRANS.X  ;
    HRnd_SidePIV_E.TRANS.X := This_SIDE.TRANS.X   ;
    !!!!!!!!END!!!!!!!
    ENDPROC

    PROC WELD_ALLPIV_1thru8 (string CAM_OR_NOT)
    !!!!!!OK FOR PTL 08-13-18

	 IF PIVOT_USED = 6089330 OR PIVOT_USED = 6802774 OR PIVOT_USED = 6870131 OR PIVOT_USED = 6845931 THEN
     !!  THIS IS FOR A 42H, 33H AND 24H
	    pivCAM := FALSE;

     ELSEIF PIVOT_USED = 6099018  OR PIVOT_USED = 674961 OR PIVOT_USED = 350404  THEN
     !!  THIS IS FOR 77F THRU 120F AND 18H !
        pivCAM := TRUE;

	ELSE STOP;

	ENDIF

	WAITTIME\INPOS,.1;

	IF CAM_OR_NOT = "G" AND pivCAM = TRUE THEN
		GOTO WELD_GCAM_1thru8;

	ELSEIF CAM_OR_NOT = "G" AND pivCAM = FALSE THEN
		GOTO WELD_GRND_1thru8;

	ELSEIF CAM_OR_NOT = "H" AND pivCAM = TRUE THEN
		GOTO WELD_HCAM_1thru8;

	ELSEIF CAM_OR_NOT = "H" AND pivCAM = FALSE THEN
		GOTO WELD_HRND_1thru8;

    ELSE STOP;

	ENDIF

 WELD_GCAM_1thru8:
        ActUnit STN1;
        BEGIN_TEST_WELD_GCAM_1thru8:
        PivGX18_Cam_18_R1 Mx_weld_piv;
        MoveJ offs(SP_gPivCam_18_Ys,600,-600,150), V500, z10, tWeldGun\WObj:=wobjHsideplate;
        MoveL offs(SP_gPivCam_18_Ys,450,100,150), V500, z10, tWeldGun\WObj:=wobjHsideplate;
        MoveL offs(SP_gPivCam_18_Ys,0,50,0), V500, z5, tWeldGun\WObj:=wobjHsideplate;
        Search_1D SR_Piv_Y\SearchStop:=PivFOUND_Y, SP_GPivCAM_18_Ys, SP_GPivCAM_18_Ye, v300, tWeldGun\WObj:=wobjHsideplate\SchSpeed:=10;
  		MoveL PivFOUND_Y, V500, z1, tWeldGun\WObj:=wobjHsideplate;
        WaitTime\InPos, 1;
        PivFOUND_Y := CRobT(\Tool:=tWeldgun\WObj:=obSTN1);
        WaitTime\InPos, 1;
        MoveL offs(SP_gPivCam_18_Ys,0,50,0), V500, z5, tWeldGun\WObj:=wobjHsideplate;
        MoveL Offs(SP_GPivCAM_18_Ys,400,100,150), V500, fine, tWeldGun\WObj:=wobjHsideplate;
        MoveJ Offs(SP_GPivCAM_18_Ys,400,-600,150), V500, z10, tWeldGun\WObj:=wobjHsideplate;
        MoveJ offs(SP_gPivCam_18_Zs,0,-200,50), v400, z10, tWeldGun\WObj:=wobjHsideplate;
        Search_1D SR_Piv_Z\SearchStop:=PivFOUND_Z, SP_GPivCAM_18_Zs, SP_GPivCAM_18_Ze, v300, tWeldGun\WObj:=wobjHsideplate\PrePDisp:=SR_Piv_Y\SchSpeed:=10;
  		MoveL PivFOUND_Z, V500, z1, tWeldGun\WObj:=wobjHsideplate;
        WaitTime\InPos, 1;
        PivFOUND_Z := CRobT(\Tool:=tWeldgun\WObj:=obSTN1);
        WaitTime\InPos, 1;
        PivWobj_Translation_Locator wobj_PivCam, PivFOUND_Y, PivFOUND_Z, WPIVOTANGLE;
        WaitTime\InPos, 1;
        MoveJ offs(SP_gPivCam_18_Zs,0, 0, 25), V500, z5, tWeldGun\WObj:=wobjHsideplate;
        MoveJ reltool(SP_gPivCam_18_Zs,0, 0, -250), V500, z10, tWeldGun\WObj:=wobjHsideplate;
        MoveJ reltool(G_CAM_1,0, 0, -150), V500, z10, tWeldGun\WObj:=wobj_PivCam;
        ArcLStart G_CAM_1, v100, smGH1thru8, wdGH1thru8\Weave:=wvGH1thru8, z1, tWeldGun\WObj:=wobj_PivCam;
		ArcL G_CAM_2, v100, smGH1thru8, wdGH1thru8\Weave:=wvGH1thru8, z1, tWeldGun\WObj:=wobj_PivCam;
		ArcL G_CAM_3, v100, smGH1thru8, wdGH1thru8\Weave:=wvGH1thru8, z5, tWeldGun\WObj:=wobj_PivCam;
		ArcL G_CAM_4, v100, smGH1thru8, wdGH1thru8\Weave:=wvGH1thru8, z5, tWeldGun\WObj:=wobj_PivCam;
		ArcL G_CAM_5, v100, smGH1thru8, wdGH1thru8\Weave:=wvGH1thru8, z5, tWeldGun\WObj:=wobj_PivCam;
		ArcL G_CAM_6, v100, smGH1thru8, wdGH1thru8\Weave:=wvGH1thru8, z5, tWeldGun\WObj:=wobj_PivCam;
		ArcL G_CAM_7, v100, smGH1thru8, wdGH1thru8\Weave:=wvGH1thru8, z5, tWeldGun\WObj:=wobj_PivCam;
        ArcLEnd G_CAM_8, v100, smGH1thru8, wdGH1thru8\Weave:=wvGH1thru8, z1, tWeldGun\WObj:=wobj_PivCam;
        MoveL reltool(G_CAM_7,0, 0, -150), V500, z10, tWeldGun\WObj:=wobj_PivCam;
		GOTO DONE_WELDING_PIV;
 WELD_HCAM_1thru8:
  	    ActUnit STN1;
        BEGIN_TEST_WELD_HCAM_1thru8:
        PivHX18_Cam_18_R1 Lx_weld_piv;
        MoveJ offs(SP_hPivCam_18_Ys,200,-300,150), V500, z10, tWeldGun\WObj:=wobjHsideplate;
        MoveL offs(SP_hPivCam_18_Ys,250,20,0), V500, z10, tWeldGun\WObj:=wobjHsideplate;
        MoveL offs(SP_hPivCam_18_Ys,0,50,0), V500, z5, tWeldGun\WObj:=wobjHsideplate;
        Search_1D SR_Piv_Y\SearchStop:=PivFOUND_Y, SP_HPivCam_18_Ys, SP_HPivCam_18_Ye, v300, tWeldGun\WObj:=wobjHsideplate\SchSpeed:=10;
  		MoveL PivFOUND_Y, V500, z1, tWeldGun\WObj:=wobjHsideplate;
        WaitTime\InPos, 1;
        PivFOUND_Y := CRobT(\Tool:=tWeldgun\WObj:=obSTN1);
        WaitTime\InPos, 1;
        MoveL offs(SP_hPivCam_18_Ys,0,50,0), V500, z5, tWeldGun\WObj:=wobjHsideplate;
        MoveL offs(SP_hPivCam_18_Ys,250,20,0), V500, z10, tWeldGun\WObj:=wobjHsideplate;
        MoveJ offs(SP_hPivCam_18_Ys,200,-300,150), V500, z10, tWeldGun\WObj:=wobjHsideplate;
        MoveJ offs(SP_hPivCam_18_Zs,100,-100,50), v400, z10, tWeldGun\WObj:=wobjHsideplate;
        Search_1D SR_Piv_Z\SearchStop:=PivFOUND_Z, SP_HPivCam_18_Zs, SP_HPivCam_18_Ze, v300, tWeldGun\WObj:=wobjHsideplate\PrePDisp:=SR_Piv_Y\SchSpeed:=10;
  		MoveL PivFOUND_Z, V500, z1, tWeldGun\WObj:=wobjHsideplate;
        WaitTime\InPos, 1;
        PivFOUND_Z := CRobT(\Tool:=tWeldgun\WObj:=obSTN1);
        WaitTime\InPos, 1;
        PivWobj_Translation_Locator wobj_PivCam, PivFOUND_Y, PivFOUND_Z, WPIVOTANGLE;
        WaitTime\InPos, 1;
        MoveJ offs(SP_hPivCam_18_Zs,0, 0, 25), V500, z5, tWeldGun\WObj:=wobjHsideplate;
        MoveJ reltool(SP_hPivCam_18_Zs,0, 0, -250), V500, z10, tWeldGun\WObj:=wobjHsideplate;
        MoveJ reltool(H_CAM_1,0, 0, -150), V500, z10, tWeldGun\WObj:=wobj_PivCam;
        ArcLStart H_CAM_1, v100, smGH1thru8, wdGH1thru8\Weave:=wvGH1thru8, z1, tWeldGun\WObj:=wobj_PivCam;
		ArcL H_CAM_2, v100, smGH1thru8, wdGH1thru8\Weave:=wvGH1thru8, z1, tWeldGun\WObj:=wobj_PivCam;
		ArcL H_CAM_3, v100, smGH1thru8, wdGH1thru8\Weave:=wvGH1thru8, z5, tWeldGun\WObj:=wobj_PivCam;
		ArcL H_CAM_4, v100, smGH1thru8, wdGH1thru8\Weave:=wvGH1thru8, z5, tWeldGun\WObj:=wobj_PivCam;
		ArcL H_CAM_5, v100, smGH1thru8, wdGH1thru8\Weave:=wvGH1thru8, z5, tWeldGun\WObj:=wobj_PivCam;
		ArcL H_CAM_6, v100, smGH1thru8, wdGH1thru8\Weave:=wvGH1thru8, z5, tWeldGun\WObj:=wobj_PivCam;
		ArcL H_CAM_7, v100, smGH1thru8, wdGH1thru8\Weave:=wvGH1thru8, z5, tWeldGun\WObj:=wobj_PivCam;
        ArcLEnd H_CAM_8, v100, smGH1thru8, wdGH1thru8\Weave:=wvGH1thru8, z1, tWeldGun\WObj:=wobj_PivCam;
        MoveL RelTool(H_CAM_8,0,0,-150), V500, z10, tWeldGun\WObj:=wobj_PivCam;
		GOTO DONE_WELDING_PIV;
WELD_GRND_1thru8:
  	    ActUnit STN1;
        BEGIN_TEST_WELD_GRND_1thru8:
        MoveJ offs(SP_gPivRnd_18_Ys,-200,-200,50), V500, z10, tWeldGun\WObj:=wobjHsideplate;
        MoveL offs(SP_gPivRnd_18_Ys,-150,25,0), V500, z10, tWeldGun\WObj:=wobjHsideplate;
        MoveL offs(SP_gPivRnd_18_Ys,0,25,0), V500, z5, tWeldGun\WObj:=wobjHsideplate;
        Search_1D SR_Piv_Y\SearchStop:=PivFOUND_Y, SP_GPivRND_18_Ys, SP_GPivRND_18_Ye, v300, tWeldGun\WObj:=wobjHsideplate\SchSpeed:=10;
  		MoveL PivFOUND_Y, V500, z1, tWeldGun\WObj:=wobjHsideplate;
        WaitTime\InPos, 1;
        PivFOUND_Y := CRobT(\Tool:=tWeldgun\WObj:=obSTN1);
        WaitTime\InPos, 1;
        MoveL offs(SP_gPivRnd_18_Ys,0,30,0), V500, z5, tWeldGun\WObj:=wobjHsideplate;
        MoveL offs(SP_gPivRnd_18_Ys,-150,30,0), V500, z5, tWeldGun\WObj:=wobjHsideplate;
        MoveL offs(SP_gPivRnd_18_Ys,-150,-400,0), V500, z10, tWeldGun\WObj:=wobjHsideplate;
        MoveJ offs(SP_gPivRnd_18_Zs,0,-200,50), v400, z10, tWeldGun\WObj:=wobjHsideplate;
        Search_1D SR_Piv_Z\SearchStop:=PivFOUND_Z, SP_gPivRnd_18_Zs, SP_gPivRnd_18_Ze, v300, tWeldGun\WObj:=wobjHsideplate\SchSpeed:=10;
  		MoveL PivFOUND_Z, V500, z1, tWeldGun\WObj:=wobjHsideplate;
        WaitTime\InPos, 1;
        PivFOUND_Z := CRobT(\Tool:=tWeldgun\WObj:=obSTN1);
        WaitTime\InPos, 1;
        PivWobj_Translation_Locator wobj_PivCam, PivFOUND_Y, PivFOUND_Z, WPIVOTANGLE;
        WaitTime\InPos, 1;
        MoveJ offs(SP_gPivRnd_18_Zs,0, 0, 25), V500, z5, tWeldGun\WObj:=wobjHsideplate;
        MoveJ reltool(SP_gPivRnd_18_Zs,-100, 0, -350), V500, z10, tWeldGun\WObj:=wobjHsideplate;
        MoveJ reltool(G_RND_1,0, 0, -350), V500, z5, tWeldGun\WObj:=wobj_PivCam;
        MoveL reltool(G_RND_1,0, 0, -100), V500, z5, tWeldGun\WObj:=wobj_PivCam;
  	    ArcLStart G_RND_1, v100, smGH1thru8, wdGH1thru8\Weave:=wvGH1thru8, z1, tWeldGun\WObj:=wobj_PivCam;
		ArcL G_RND_2, v100, smGH1thru8, wdGH1thru8\Weave:=wvGH1thru8, z1, tWeldGun\WObj:=wobj_PivCam;
		ArcL G_RND_3, v100, smGH1thru8, wdGH1thru8\Weave:=wvGH1thru8, z1, tWeldGun\WObj:=wobj_PivCam;
		ArcL G_RND_4, v100, smGH1thru8, wdGH1thru8\Weave:=wvGH1thru8, z1, tWeldGun\WObj:=wobj_PivCam;
		ArcL G_RND_5, v100, smGH1thru8, wdGH1thru8\Weave:=wvGH1thru8, z1, tWeldGun\WObj:=wobj_PivCam;
        ArcLEnd G_RND_6, v100, smGH1thru8, wdGH1thru8\Weave:=wvGH1thru8, z1, tWeldGun\WObj:=wobj_PivCam;
        MoveL reltool(G_RND_6,0, 0, -100), V500, z10, tWeldGun\WObj:=wobj_PivCam;
        MoveL reltool(G_RND_7,0, 0, -100), V500, z10, tWeldGun\WObj:=wobj_PivCam;
        GOTO DONE_WELDING_PIV;
WELD_HRND_1thru8:
  	    ActUnit STN1;
        BEGIN_TEST_WELD_HRND_1thru8:
        MoveJ offs(SP_HPivRND_18_Ys,200,50,50), V500, z10, tWeldGun\WObj:=wobjHsideplate;
        MoveL offs(SP_HPivRND_18_Ys,150,75,50), V500, z10, tWeldGun\WObj:=wobjHsideplate;
        MoveL offs(SP_HPivRND_18_Ys,0,50,0), V500, z5, tWeldGun\WObj:=wobjHsideplate;
        Search_1D SR_Piv_Y\SearchStop:=PivFOUND_Y, SP_HPivRND_18_Ys, SP_HPivRND_18_Ye, v300, tWeldGun\WObj:=wobjHsideplate\SchSpeed:=10;
  		MoveL PivFOUND_Y, V500, z1, tWeldGun\WObj:=wobjHsideplate;
        WaitTime\InPos, 1;
        PivFOUND_Y := CRobT(\Tool:=tWeldgun\WObj:=obSTN1);
        WaitTime\InPos, 1;
        MoveL offs(SP_HPivRND_18_Ys,0,50,0), V500, z5, tWeldGun\WObj:=wobjHsideplate;
        MoveL offs(SP_HPivRND_18_Ys,150,75,50), V500, z10, tWeldGun\WObj:=wobjHsideplate;
        MoveL offs(SP_HPivRND_18_Ys,150,-450,50), V500, z10, tWeldGun\WObj:=wobjHsideplate;
        MoveJ offs(SP_HPivRND_18_Zs,150,-100,50), v400, z10, tWeldGun\WObj:=wobjHsideplate;
        MoveL offs(SP_HPivRND_18_Zs,0,0,50), v400, z10, tWeldGun\WObj:=wobjHsideplate;
        Search_1D SR_Piv_Z\SearchStop:=PivFOUND_Z, SP_HPivRND_18_Zs, SP_HPivRND_18_Ze, v300, tWeldGun\WObj:=wobjHsideplate\SchSpeed:=10;
  		MoveL PivFOUND_Z, V500, z1, tWeldGun\WObj:=wobjHsideplate;
        WaitTime\InPos, 1;
        PivFOUND_Z := CRobT(\Tool:=tWeldgun\WObj:=obSTN1);
        WaitTime\InPos, 1;
        PivWobj_Translation_Locator wobj_PivCam, PivFOUND_Y, PivFOUND_Z, WPIVOTANGLE;
        WaitTime\InPos, 1;
        MoveL offs(SP_HPivRND_18_Zs,0, 0, 25), V500, z5, tWeldGun\WObj:=wobjHsideplate;
        MoveL offs(SP_HPivRND_18_Zs,75, -350, 25), V500, z5, tWeldGun\WObj:=wobjHsideplate;
        MoveJ reltool(H_RND_1,0, 0, -150), V500, z10, tWeldGun\WObj:=wobj_PivCam;
        ArcLStart H_RND_1, v100, smGH1thru8, wdGH1thru8\Weave:=wvGH1thru8, z1, tWeldGun\WObj:=wobj_PivCam;
		ArcL H_RND_2, v100, smGH1thru8, wdGH1thru8\Weave:=wvGH1thru8, z1, tWeldGun\WObj:=wobj_PivCam;
		ArcL H_RND_3, v100, smGH1thru8, wdGH1thru8\Weave:=wvGH1thru8, z1, tWeldGun\WObj:=wobj_PivCam;
		ArcL H_RND_4, v100, smGH1thru8, wdGH1thru8\Weave:=wvGH1thru8, z1, tWeldGun\WObj:=wobj_PivCam;
		ArcL H_RND_5, v100, smGH1thru8, wdGH1thru8\Weave:=wvGH1thru8, z1, tWeldGun\WObj:=wobj_PivCam;
        ArcLEnd H_RND_6, v100, smGH1thru8, wdGH1thru8\Weave:=wvGH1thru8, z1, tWeldGun\WObj:=wobj_PivCam;
        MoveL reltool(H_RND_6,0, 0, -100), V500, z10, tWeldGun\WObj:=wobj_PivCam;
        MoveL reltool(H_RND_7,0, 0, -100), V500, z10, tWeldGun\WObj:=wobj_PivCam;
        !GOTO DONE_WELDING_PIV;
    	DONE_WELDING_PIV:
    ENDPROC

    PROC WELD_ALLPIV_PJ_18H (string RND_OR_CAM)
      !!!!OK FOR PTL 08-16-18!!!
	 IF PIVOT_USED = 6089330 OR PIVOT_USED = 6802774 OR PIVOT_USED = 6870131 OR PIVOT_USED = 6845931 THEN
     !!  THIS IS FOR A 42H, 33H AND 24H
	    pivCAM := FALSE;

 	ELSEIF PIVOT_USED =  674961 OR PIVOT_USED = 350404 OR PIVOT_USED = 6099018 THEN
     !!  THIS IS FOR 77F THRU 120F AND 18H !
        pivCAM := TRUE;

	ELSE STOP;

	ENDIF

	WAITTIME\INPOS,.1;

	IF RND_OR_CAM = "G" AND pivCAM = TRUE THEN
		GOTO WELD_GCAM_PJ;

	ELSEIF RND_OR_CAM = "G" AND pivCAM = FALSE THEN
		GOTO WELD_GRND_PJ;

	ELSEIF RND_OR_CAM = "H" AND pivCAM = TRUE THEN
		GOTO WELD_HCAM_PJ;

	ELSEIF RND_OR_CAM = "H" AND pivCAM = FALSE THEN
		GOTO WELD_HRND_PJ;

    ELSE STOP;

	ENDIF

 WELD_GCAM_PJ:
        ActUnit STN1;
        BEGIN_TEST_WELD_GCAM_PJ:
        ActUnit STN1;
        MoveJ pjthomeSTA1zero, vCellSpeed, fine, tWeldGun\WObj:=wobj0;
        MoveJ Offs(SP_gPivCam_PJ_Xs, -250, 0, 0), V500, z10, tWeldGun\WObj:=wobj_PivCam;
        MoveL Offs(SP_gPivCam_PJ_Xs, -50, 0, 0), V500, z5, tWeldGun\WObj:=wobj_PivCam;
        Search_1D SR_Gx\SearchStop:=gX_FOUND, SP_gPivCam_PJ_Xs, SP_gPivCam_PJ_Xe, v50, tWeldGun\WObj:=wobj_PivCam\SchSpeed:=10;
        MoveL Offs(SP_gPivCam_PJ_Xs, -50, 0, 0), V500, z5, tWeldGun\WObj:=wobj_PivCam;
        MoveL Offs(SP_gPivCam_PJ_Xs, -250, 0, 0), V500, z10, tWeldGun\WObj:=wobj_PivCam;
        PivGXPJ_Cam_18_R1 gX_FOUND;
        MoveJ offs(SP_gPivCam_PJ_Ys,-100,50,0), V500, z10, tWeldGun\WObj:=wobjHsideplate;
        MoveL offs(SP_gPivCam_PJ_Ys,0,50,0), V500, z5, tWeldGun\WObj:=wobjHsideplate;
        Search_1D SR_Piv_Y\SearchStop:=PivFOUND_Y, SP_GPivCAM_PJ_Ys, SP_GPivCAM_PJ_Ye, v300, tWeldGun\WObj:=wobjHsideplate\SchSpeed:=10;
  		MoveL PivFOUND_Y, V500, z1, tWeldGun\WObj:=wobjHsideplate;
        WaitTime\InPos, 1;
        PivFOUND_Y := CRobT(\Tool:=tWeldgun\WObj:=obSTN1);
        WaitTime\InPos, 1;
        MoveL offs(SP_gPivCam_PJ_Ys,-50,50,0), V500, z5, tWeldGun\WObj:=wobjHsideplate;
        MoveL offs(SP_gPivCam_PJ_Ys,-150,50,0), V500, z10, tWeldGun\WObj:=wobjHsideplate;
        MoveJ offs(SP_gPivCam_PJ_Zs,-150,-50,50), V500, z10, tWeldGun\WObj:=wobjHsideplate;
        MoveL offs(SP_gPivCam_PJ_Zs,0,0,50), v400, z10, tWeldGun\WObj:=wobjHsideplate;
        Search_1D SR_Piv_Z\SearchStop:=PivFOUND_Z, SP_GPivCAM_PJ_Zs, SP_GPivCAM_PJ_Ze, v300, tWeldGun\WObj:=wobjHsideplate\PrePDisp:=SR_Piv_Y\SchSpeed:=10;
  		MoveL PivFOUND_Z, V500, z1, tWeldGun\WObj:=wobjHsideplate;
        WaitTime\InPos, 1;
        PivFOUND_Z := CRobT(\Tool:=tWeldgun\WObj:=obSTN1);
        WaitTime\InPos, 1;
        PivWobj_Translation_Locator wobj_PivCam, PivFOUND_Y, PivFOUND_Z, WPIVOTANGLE;
        MoveJ offs(SP_gPivCam_PJ_Zs,0, 0, 25), V500, z5, tWeldGun\WObj:=wobjHsideplate;
        MoveJ offs(SP_gPivCam_PJ_Zs,-300, -50, 25), V500, z10, tWeldGun\WObj:=wobjHsideplate;
        MoveJ reltool(G_PJCam_1st_s,0, 0, -250), V500, z10, tWeldGun\WObj:=wobj_PivCam;
     	MoveL RelTool(SP_GCAM_PJEDGE_S,0,0,-20), v100, z1, tWeldGun\WObj:=wobj_PivCam;
   		Search_Edge\TopCornerDisp:=SRG_PJ_EDGE, SP_GCAM_PjEDGE_S, SP_GCAM_PjEDGE_E, edgedata_GCAM_PJ\InitSchL:=15\Spacing:=3\PackStart, v50, tWeldGun\WObj:=wobj_PivCam\SrchSpeed:=5;
        TPWrite "SRG_PJ_EDGE XYZ:="\Pos:=SRG_PJ_EDGE.trans;
        MoveL RelTool(SP_GCAM_PJEDGE_S,0,0,-20), v100, z1, tWeldGun\WObj:=wobj_PivCam;
		Search_Joint SRG_PJ_JOINT, SP_GCAM_PjJOINT_S, SP_GCAM_PjJOINT_E, bevelparam_GCAM_PJ, seampar_GCAM_PJ\InitSchL:=15\PackStart, v50, tWeldGun\WObj:=wobj_PivCam\PrePDisp:=SRG_PJ_EDGE\SrchSpeed:=5;
		MoveL RelTool(G_PJCam_1st_S,0,0,-100), v100, z1, tWeldGun\WObj:=wobj_PivCam;
        TPWrite "SRG_PJ_JOINT XYZ:="\Pos:=SRG_PJ_JOINT.trans;
        SRG_PJ_EDGE.trans.x := 0;
        SRG_PJ_JOINT.trans.x := 0;
        TPWrite "mm2 Weld Area Calculated:="\num:=seampar_GCAM_PJ.Area;
        TPWrite "NOW WORKING ON 'GCAM'(Root Pass)";
        !the percentages in this IF affect the G root pass only!
        IF seampar_GCAM_PJ.Area < 175 THEN
    	seampar_GCAM_PJ.Weldpar.fill_pct := percentrootpass;
        ELSEIF   seampar_GCAM_PJ.Area > 175  and seampar_GCAM_PJ.Area < 475 THEN
    	seampar_GCAM_PJ.Weldpar.fill_pct := percentrootpass;
        ELSEIF seampar_GCAM_PJ.Area > 475 THEN
    	seampar_GCAM_PJ.Weldpar.fill_pct := percentrootpass;
        ENDIF
		weldin_now:
	    IF bWO455only = TRUE OR bWO456only = TRUE THEN   seampar_GCAM_PJ.Weldpar.wirefeed:=(wdGH_CAM_PJ_ROOT.main_arc.wirefeed *60)/25.4;
	    ENDIF
	    IF bWO458only = TRUE OR bWO459only = TRUE THEN   seampar_GCAM_PJ.Weldpar.wirefeed:=wdGH_CAM_PJ_ROOT.main_arc.wirefeed;
	    ENDIF
        PDispSet SRG_PJ_EDGE;
		HWeldStart G_PJCam_1st_S, seampar_GCAM_PJ, smGH_RND_PJ, wdGH_CAM_PJ_ROOT\Weave:=wv0, v100, z1, tWeldGun\WObj:=wobj_PivCam;
        TPWrite "G Root Pass fill percentage:="\Num:=seampar_GCAM_PJ.Weldpar.fill_pct;
		TPWrite "seampar_GCAM_PJ Wirefeed:="\num:=seampar_GCAM_PJ.Weldpar.wirefeed;
		WaitTime 0.75;
		HWeldL G_PJCam_1st_SM,seampar_GCAM_PJ, v100, z1, tWeldGun\WObj:=wobj_PivCam;
		HWeldL G_PJCam_1st_EM,seampar_GCAM_PJ, v100, z1, tWeldGun\WObj:=wobj_PivCam;
		HWeldLEnd G_PJCam_1st_E,seampar_GCAM_PJ, v100,  z1, tWeldGun\WObj:=wobj_PivCam;
		MoveL RelTool(G_PJCam_1st_S,0,0,-100), v100, z1, tWeldGun\WObj:=wobj_PivCam;
		PDispOff;
        G_NOMINAL:
		seampar_GCAM_PJ.Weldpar.fill_pct := percent2pass;
	    IF bWO455only = TRUE OR bWO456only = TRUE THEN   seampar_GCAM_PJ.Weldpar.wirefeed:=(wdGH_CAM_PJ_CVR.main_arc.wirefeed *60)/25.4;
	    ENDIF
	    IF bWO458only = TRUE OR bWO459only = TRUE THEN   seampar_GCAM_PJ.Weldpar.wirefeed:=wdGH_CAM_PJ_CVR.main_arc.wirefeed;
	    ENDIF
        TPWrite "NOW WORKING ON Nominal 'G50'(Final pass)";
        TPWrite "G Final Pass fill percentage:="\Num:=seampar_GCAM_PJ.Weldpar.fill_pct;
        WaitTime 5;
		PDispSet SRG_PJ_JOINT;
		HWeldStart G_PJCam_4th_E, seampar_GCAM_PJ, smGH_CAM_PJ, wdGH_CAM_PJ_CVR\Weave:=wvGH_CAM_PJ_CVR, v100, z1, tWeldGun\WObj:=wobj_PivCam;
		HWeldL G_PJCam_4th_EM, seampar_GCAM_PJ, v100, z1, tWeldGun\WObj:=wobj_PivCam;
		HWeldL G_PJCam_4th_SM, seampar_GCAM_PJ, v100, z1, tWeldGun\WObj:=wobj_PivCam;
		HWeldLEnd G_PJCam_4th_S, seampar_GCAM_PJ, v100, z1, tWeldGun\WObj:=wobj_PivCam;
        TPErase;
		PDispOff;
		MoveL RelTool(G_PJCam_2nd_S,0,0,-250), v300, z1, tWeldGun\WObj:=wobj_PivCam;
		GOTO DONE_WELDING_PJ;
 WELD_HCAM_PJ:
        ActUnit STN1;
        BEGIN_TEST_WELD_HCAM_PJ:
        MoveJ pjthomeSTA1zero, vCellSpeed, fine, tWeldGun\WObj:=wobj0;
        MoveJ Offs(SP_hPivCam_PJ_Xs,200, 0, 0), V500, z10, tWeldGun\WObj:=wobj_PivCam;
        MoveL offs(SP_hPivCam_PJ_Xs, 50, 0, 0), V500, z5, tWeldGun\WObj:=wobj_PivCam;
        Search_1D SR_Hx\SearchStop:=hX_FOUND, SP_hPivCam_PJ_Xs, SP_hPivCam_PJ_Xe, v50, tWeldGun\WObj:=wobj_PivCam\SchSpeed:=10;
        MoveL offs(SP_hPivCam_PJ_Xs, 50, 0, 0), V500, z5, tWeldGun\WObj:=wobj_PivCam;
        MoveL Offs(SP_hPivCam_PJ_Xs,200, 0, 0), V500, z10, tWeldGun\WObj:=wobj_PivCam;
        PivHXPJ_Cam_18_R1 hX_FOUND;
        MoveJ offs(SP_hPivCam_PJ_Ys,150,50,00), V500, z10, tWeldGun\WObj:=wobjHsideplate;
        MoveL offs(SP_hPivCam_PJ_Ys,0,50,0), V500, z10, tWeldGun\WObj:=wobjHsideplate;
        MoveL offs(SP_hPivCam_PJ_Ys,0,50,0), V500, z5, tWeldGun\WObj:=wobjHsideplate;
        Search_1D SR_Piv_Y\SearchStop:=PivFOUND_Y, SP_HPivCam_PJ_Ys, SP_HPivCam_PJ_Ye, v300, tWeldGun\WObj:=wobjHsideplate\SchSpeed:=10;
  		MoveL PivFOUND_Y, V500, z1, tWeldGun\WObj:=wobjHsideplate;
        WaitTime\InPos, 1;
        PivFOUND_Y := CRobT(\Tool:=tWeldgun\WObj:=obSTN1);
        WaitTime\InPos, 1;
        MoveL offs(SP_hPivCam_PJ_Ys,0,50,0), V500, z5, tWeldGun\WObj:=wobjHsideplate;
        MoveL offs(SP_hPivCam_PJ_Ys,150,100,0), V500, z10, tWeldGun\WObj:=wobjHsideplate;
        MoveJ offs(SP_hPivCam_PJ_Zs,150,50,25), V500, z10, tWeldGun\WObj:=wobjHsideplate;
        MoveJ offs(SP_hPivCam_PJ_Zs,0,0,50), v400, z10, tWeldGun\WObj:=wobjHsideplate;
        Search_1D SR_Piv_Z\SearchStop:=PivFOUND_Z, SP_HPivCam_PJ_Zs, SP_HPivCam_PJ_Ze, v300, tWeldGun\WObj:=wobjHsideplate\PrePDisp:=SR_Piv_Y\SchSpeed:=10;
  		MoveL PivFOUND_Z, V500, z1, tWeldGun\WObj:=wobjHsideplate;
        WaitTime\InPos, 1;
        PivFOUND_Z := CRobT(\Tool:=tWeldgun\WObj:=obSTN1);
        WaitTime\InPos, 1;
        PivWobj_Translation_Locator wobj_PivCam, PivFOUND_Y, PivFOUND_Z, WPIVOTANGLE;
        MoveJ offs(SP_hPivCam_PJ_Zs,0, 0, 25), V500, z5, tWeldGun\WObj:=wobjHsideplate;
        MoveJ offs(SP_hPivCam_PJ_Zs,200, 0, 25), V500, z10, tWeldGun\WObj:=wobjHsideplate;
        MoveJ reltool(SP_HCAM_PJEDGE_s,0, 0, -250), V500, z10, tWeldGun\WObj:=wobj_PivCam;
        MoveL reltool(SP_HCAM_PJEDGE_s,0, 0, -50), V500, z10, tWeldGun\WObj:=wobj_PivCam;
     	MoveL RelTool(SP_HCAM_PJEDGE_S,0,0,-20), v100, z1, tWeldGun\WObj:=wobj_PivCam;
		Search_Edge\TopCornerDisp:=SRH_PJ_EDGE, SP_HCAM_PjEDGE_S, SP_HCAM_PjEDGE_E, edgedata_HCAM_PJ\InitSchL:=15\Spacing:=3\PackStart, v50, tWeldGun\WObj:=wobj_PivCam\SrchSpeed:=5;
        TPWrite "SRH_PJ_EDGE XYZ:="\Pos:=SRH_PJ_EDGE.trans;
        MoveL RelTool(SP_HCAM_PJEDGE_S,0,0,-20), v100, z1, tWeldGun\WObj:=wobj_PivCam;
		Search_Joint SRH_PJ_JOINT, SP_HCAM_PjJOINT_S, SP_HCAM_PjJOINT_E, bevelparam_HCAM_PJ, seampar_HCAM_PJ\InitSchL:=15\PackStart, v50, tWeldGun\WObj:=wobj_PivCam\PrePDisp:=SRH_PJ_EDGE\SrchSpeed:=5;
		MoveL RelTool(H_PJCam_1st_S,0,0,-100), v100, z1, tWeldGun\WObj:=wobj_PivCam;
        TPWrite "SRH_PJ_JOINT XYZ:="\Pos:=SRH_PJ_JOINT.trans;
        TPWrite "mm2 Weld Area Calculated:="\num:=seampar_HCAM_PJ.Area;
        SRH_PJ_EDGE.trans.x := 0;
        SRH_PJ_JOINT.trans.x := 0;
        TPWrite "NOW WORKING ON 'HCAM'(Root Pass)";
        !the percentages in this IF affect the H root pass only!
        IF seampar_HCAM_PJ.Area < 175 THEN
    	seampar_HCAM_PJ.Weldpar.fill_pct := percentrootpass;
        ELSEIF   seampar_HCAM_PJ.Area > 175  and seampar_HCAM_PJ.Area < 475 THEN
    	seampar_HCAM_PJ.Weldpar.fill_pct := percentrootpass;
        ELSEIF seampar_HCAM_PJ.Area > 475 THEN
    	seampar_HCAM_PJ.Weldpar.fill_pct := percentrootpass;
        ENDIF
        weldin_H_now:
	    IF bWO455only = TRUE OR bWO456only = TRUE THEN   seampar_HCAM_PJ.Weldpar.wirefeed:=(wdGH_CAM_PJ_ROOT.main_arc.wirefeed *60)/25.4;
	    ENDIF
	    IF bWO458only = TRUE OR bWO459only = TRUE THEN   seampar_HCAM_PJ.Weldpar.wirefeed:=wdGH_CAM_PJ_ROOT.main_arc.wirefeed;
	    ENDIF
        PDispSet SRH_PJ_EDGE;
		HWeldStart H_PJCam_1st_S, seampar_HCAM_PJ, smGH_RND_PJ, wdGH_CAM_PJ_ROOT\Weave:=wv0, v100, z1, tWeldGun\WObj:=wobj_PivCam;
        TPWrite "H Root Pass fill percentage:="\Num:=seampar_HCAM_PJ.Weldpar.fill_pct;
		TPWrite "seampar_HCAM_PJ Wirefeed:="\num:=seampar_HCAM_PJ.Weldpar.wirefeed;
		WaitTime 0.75;
		HWeldL H_PJCam_1st_SM,seampar_HCAM_PJ, v100, z1, tWeldGun\WObj:=wobj_PivCam;
		HWeldL H_PJCam_1st_EM,seampar_HCAM_PJ, v100, z1, tWeldGun\WObj:=wobj_PivCam;
		HWeldLEnd H_PJCam_1st_E,seampar_HCAM_PJ, v100,  z1, tWeldGun\WObj:=wobj_PivCam;
		MoveL RelTool(H_PJCam_1st_S,0,0,-100), v100, z1, tWeldGun\WObj:=wobj_PivCam;
		PDispOff;
    H_NOMINAL:
		seampar_HCAM_PJ.Weldpar.fill_pct := percent2pass;
	    IF bWO455only = TRUE OR bWO456only = TRUE THEN   seampar_GCAM_PJ.Weldpar.wirefeed:=(wdGH_CAM_PJ_CVR.main_arc.wirefeed *60)/25.4;
	    ENDIF
	    IF bWO458only = TRUE OR bWO459only = TRUE THEN   seampar_GCAM_PJ.Weldpar.wirefeed:=wdGH_CAM_PJ_CVR.main_arc.wirefeed;
	    ENDIF
        TPWrite "NOW WORKING ON Nominal 'G50'(Final pass)";
        TPWrite "G Final Pass fill percentage:="\Num:=seampar_HCAM_PJ.Weldpar.fill_pct;
        WaitTime 5;
		PDispSet SRH_PJ_JOINT;
		HWeldStart H_PJCam_4th_E, seampar_HCAM_PJ, smGH_CAM_PJ, wdGH_CAM_PJ_CVR\Weave:=wvGH_CAM_PJ_CVR, v100, z1, tWeldGun\WObj:=wobj_PivCam;
		HWeldL H_PJCam_4th_EM, seampar_HCAM_PJ, v100, z1, tWeldGun\WObj:=wobj_PivCam;
		HWeldL H_PJCam_4th_sm, seampar_HCAM_PJ, v100, z1, tWeldGun\WObj:=wobj_PivCam;
		HWeldLEnd H_PJCam_4th_S, seampar_HCAM_PJ, v100, z1, tWeldGun\WObj:=wobj_PivCam;
        TPErase;
		PDispOff;
		MoveL RelTool(H_PJCam_2nd_S,0,0,-250), v300, z1, tWeldGun\WObj:=wobj_PivCam;
		MoveJ pjthomeSTA1zero, vCellSpeed, fine, tWeldGun\WObj:=wobj0;
		GOTO DONE_WELDING_PJ;
WELD_GRND_PJ:
     	ActUnit STN1;
        BEGIN_TEST_WELD_GRND_PJ:
        ActUnit STN1;
        MoveJ pjthomeSTA1zero, vCellSpeed, fine, tWeldGun\WObj:=wobj0;
        MoveJ OFFS(SP_gPivRnd_PJ_Xs, 350, -150, 0), V500, z10, tWeldGun\ WObj:=wobj_PivCam;
        MoveL OFFS(SP_gPivRnd_PJ_Xs, 100, -150, 0), V500, z10, tWeldGun\WObj:=wobj_PivCam;
        MoveL OFFS(SP_gPivRnd_PJ_Xs, 10, 0, 0), V500, z5, tWeldGun\WObj:=wobj_PivCam;
        Search_1D SR_Gx\SearchStop:=gX_FOUND, SP_gPivRnd_PJ_Xs, SP_gPivRnd_PJ_Xe, v50, tWeldGun\WObj:=wobj_PivCam\SchSpeed:=10;
        MoveL RelTooL(SP_gPivRnd_PJ_Xs, 0, 0, -50), V500, z5, tWeldGun\WObj:=wobj_PivCam;
        MoveL OFFS(SP_gPivRnd_PJ_Xs, 100, -200, 0), V500, z10, tWeldGun\WObj:=wobj_PivCam;
        MoveL OFFS(SP_gPivRnd_PJ_Xs, 450, -150, 0), V500, z10, tWeldGun\ WObj:=wobj_PivCam;
        PivGXPJ_Rnd gX_FOUND;
        MoveJ offs(SP_gPivRnd_PJ_Ys,600,0,150), V500, z10, tWeldGun\WObj:=wobjHsideplate;
        MoveL offs(SP_gPivRnd_PJ_Ys,600,0,150), V500, z10, tWeldGun\WObj:=wobjHsideplate;
        MoveL offs(SP_gPivRnd_PJ_Ys,450,100,150), V500, z10, tWeldGun\WObj:=wobjHsideplate;
        MoveL offs(SP_gPivRnd_PJ_Ys,0,50,0), V500, z5, tWeldGun\WObj:=wobjHsideplate;
        Search_1D SR_Piv_Y\SearchStop:=PivFOUND_Y, SP_GPivRND_PJ_Ys, SP_GPivRND_PJ_Ye, v300, tWeldGun\WObj:=wobjHsideplate\SchSpeed:=10;
  		MoveL PivFOUND_Y, V500, z1, tWeldGun\WObj:=wobjHsideplate;
        WaitTime\InPos, 1;
        PivFOUND_Y := CRobT(\Tool:=tWeldgun\WObj:=obSTN1);
        WaitTime\InPos, 1;
        MoveL offs(SP_gPivRnd_PJ_Ys,0,150,0), V500, z5, tWeldGun\WObj:=wobjHsideplate;
        MoveL offs(SP_gPivRnd_PJ_Ys,-150,150,0), V500, z5, tWeldGun\WObj:=wobjHsideplate;
        MoveL offs(SP_gPivRnd_PJ_Zs,-150,150,0), V500, z10, tWeldGun\WObj:=wobjHsideplate;
        MoveJ offs(SP_gPivRnd_PJ_Zs,0,50,50), v400, z10, tWeldGun\WObj:=wobjHsideplate;
        Search_1D SR_Piv_Z\SearchStop:=PivFOUND_Z, SP_gPivRnd_PJ_Zs, SP_gPivRnd_PJ_Ze, v300, tWeldGun\WObj:=wobjHsideplate\PrePDisp:=SR_Piv_Y\SchSpeed:=10;
  		MoveL PivFOUND_Z, V500, z1, tWeldGun\WObj:=wobjHsideplate;
        WaitTime\InPos, 1;
        PivFOUND_Z := CRobT(\Tool:=tWeldgun\WObj:=obSTN1);
        WaitTime\InPos, 1;
        PivWobj_Translation_Locator wobj_PivCam, PivFOUND_Y, PivFOUND_Z, WPIVOTANGLE;
        MoveL offs(SP_gPivRnd_PJ_Zs,0, 0, 25), V500, z5, tWeldGun\WObj:=wobjHsideplate;
        MoveL offs(SP_gPivRnd_PJ_Zs,0, 200, 25), V500, z5, tWeldGun\WObj:=wobjHsideplate;
        MoveL offs(SP_gPivRnd_PJ_Zs,600, 200, 25), V500, z10, tWeldGun\WObj:=wobjHsideplate;
        MoveJ offs(G_PJRnd_1st_s,350, -100, 0), V500, z5, tWeldGun\WObj:=wobj_PivCam;
        MoveL offs(G_PJRnd_1st_s,100, -150, 0), V500, z5, tWeldGun\WObj:=wobj_PivCam;
     	MoveL RelTool(SP_GRND_PJEDGE_S,0,0,-20), v100, z1, tWeldGun\WObj:=wobj_PivCam;
		Search_Edge\TopCornerDisp:=SRG_PJ_EDGE, SP_Grnd_PjEDGE_S, SP_Grnd_PjEDGE_E, edgedata_GRND_PJ\InitSchL:=15\Spacing:=3\PackStart, v50, tWeldGun\WObj:=wobj_PivCam\SrchSpeed:=5;
        TPWrite "SRG_PJ_EDGE XYZ:="\Pos:=SRG_PJ_EDGE.trans;
        MoveL RelTool(SP_Grnd_PJEDGE_S,0,0,-20), v100, z1, tWeldGun\WObj:=wobj_PivCam;
		Search_Joint SRG_PJ_JOINT, SP_Grnd_PjJOINT_S, SP_Grnd_PjJOINT_E, bevelparam_GRND_PJ, seampar_GRND_PJ\InitSchL:=15\PackStart, v50, tWeldGun\WObj:=wobj_PivCam\PrePDisp:=SRG_PJ_EDGE\SrchSpeed:=5;
		MoveL Offs(G_PJRnd_1st_s,30,-30,0), v100, z1, tWeldGun\WObj:=wobj_PivCam;
        TPWrite "SRG_PJ_JOINT XYZ:="\Pos:=SRG_PJ_JOINT.trans;
        TPWrite "mm2 Weld Area Calculated:="\num:=seampar_GRND_PJ.Area;
        SRG_PJ_EDGE.trans.x := 0;
        SRG_PJ_JOINT.trans.x := 0;
        TPWrite "NOW WORKING ON WELD 'GPJ_ROUND'(root)";
        seampar_GRND_PJ.Weldpar.fill_pct := percentrootpass;
	   IF bWO455only = TRUE OR bWO456only = TRUE THEN   seampar_GRND_PJ.Weldpar.wirefeed:=(wdGH_RND_PJ_CVR.main_arc.wirefeed *60)/25.4;
	    ENDIF
	    IF bWO458only = TRUE OR bWO459only = TRUE THEN   seampar_GRND_PJ.Weldpar.wirefeed:=wdGH_RND_PJ_CVR.main_arc.wirefeed;
	    ENDIF
	    PDispSet SRG_PJ_EDGE;
		HWeldStart G_PJRnd_1st_E, seampar_GRND_PJ, smGH_RND_PJ, wdGH_RND_PJ_CVR\Weave:=wv0, v100, z1, tWeldGun\WObj:=wobj_PivCam;
		HWeldL G_PJRnd_1st_EM, seampar_GRND_PJ, v100, z1, tWeldGun\WObj:=wobj_PivCam;
        HWeldLEnd G_PJRnd_1st_s, seampar_GRND_PJ, v100, z1, tWeldGun\WObj:=wobj_PivCam;
		MoveL offs(G_PJRnd_1st_s,30,-30,0), v100, z1, tWeldGun\WObj:=wobj_PivCam;
		PDispOff;
        TPWrite "NOW WORKING ON WELD 'GPJ_ROUND'(2nd pass)";
		WaitTime 4;
    	seampar_GRND_PJ.Weldpar.fill_pct := percentcoverpass;

	   IF bWO455only = TRUE OR bWO456only = TRUE THEN   seampar_GRND_PJ.Weldpar.wirefeed:=(wdGH_RND_PJ_CVR.main_arc.wirefeed *60)/25.4;
	    ENDIF
	    IF bWO458only = TRUE OR bWO459only = TRUE THEN   seampar_GRND_PJ.Weldpar.wirefeed:=wdGH_RND_PJ_CVR.main_arc.wirefeed;
	    ENDIF
		PDispSet SRG_PJ_JOINT;
		HWeldStart G_PJRnd_2nd_S, seampar_GRND_PJ, smGH_RND_PJ, wdGH_RND_PJ_CVR\Weave:=wvGH_RND_PJ_CVR, v100, z1, tWeldGun\WObj:=wobj_PivCam\Track:=trPJhiteonly1;
		HWeldL G_PJRnd_2nd_SM, seampar_GRND_PJ, v100, z1, tWeldGun\WObj:=wobj_PivCam;
		HWeldL G_PJRnd_2nd_EM, seampar_GRND_PJ, v100, z1, tWeldGun\WObj:=wobj_PivCam;
        HWeldLEnd G_PJRnd_2nd_E, seampar_GRND_PJ, v100, z1, tWeldGun\WObj:=wobj_PivCam;
        MoveL offs(G_PJRnd_1st_s,30,-30,0), v100, z1, tWeldGun\WObj:=wobj_PivCam;
        MoveL Offs(G_PJRnd_1st_s,100,-50,0), v100, z1, tWeldGun\WObj:=wobj_PivCam;
        MoveL offs(G_PJRnd_1st_s,200, -100, 0), V500, z5, tWeldGun\WObj:=wobj_PivCam;
        MoveL offs(G_PJRnd_1st_s,400, -100, 0), V500, z5, tWeldGun\WObj:=wobj_PivCam;
        MoveJ pjthomeSTA1zero, vCellSpeed, fine, tWeldGun\WObj:=wobj0;
		GOTO DONE_WELDING_PJ;
    WELD_HRND_PJ:
  	    ActUnit STN1;
        BEGIN_TEST_WELD_HRND_PJ:
        MoveJ pjthomeSTA1zero, vCellSpeed, fine, tWeldGun\WObj:=wobj0;
        MoveJ Offs(SP_hPivRND_PJ_Xs, -500, -150, 100), V500, z10, tWeldGun\WObj:=wobj_PivCam;
        MoveL Offs(SP_hPivRND_PJ_Xs, -50, -150, 100), V500, z10, tWeldGun\WObj:=wobj_PivCam;
        MoveL RelTooL(SP_hPivRND_PJ_Xs, 0, 0, -50), V500, z5, tWeldGun\WObj:=wobj_PivCam;
        Search_1D SR_Hx\SearchStop:=hX_FOUND, SP_hPivRND_PJ_Xs, SP_hPivRND_PJ_Xe, v50, tWeldGun\WObj:=wobj_PivCam\SchSpeed:=10;
        MoveL RelTooL(SP_hPivRND_PJ_Xs, 0, 0, -100), V500, z5, tWeldGun\WObj:=wobj_PivCam;
        MoveL RelTooL(SP_hPivRND_PJ_Xs, 0, 0, -200), V500, z10, tWeldGun\WObj:=wobj_PivCam;
        PivHXPJ_Rnd hX_FOUND;
        MoveJ offs(SP_HPivRND_PJ_Zs,0,-250,50), V500, z10, tWeldGun\WObj:=wobjHsideplate;
        MoveL offs(SP_HPivRND_PJ_Zs,0,-250,50), V500, z10, tWeldGun\WObj:=wobjHsideplate;
        MoveL offs(SP_HPivRND_PJ_Zs,0,0,20), V500, z5, tWeldGun\WObj:=wobjHsideplate;
        Search_1D SR_Piv_Z\SearchStop:=PivFOUND_Z, SP_HPivRND_PJ_Zs, SP_HPivRND_PJ_Ze, v300, tWeldGun\WObj:=wobjHsideplate\SchSpeed:=10;
  		MoveL PivFOUND_Z, V500, z1, tWeldGun\WObj:=wobjHsideplate;
        WaitTime\InPos, 1;
        PivFOUND_Z := CRobT(\Tool:=tWeldgun\WObj:=obSTN1);
        WaitTime\InPos, 1;
        MoveL offs(SP_HPivRND_PJ_Zs,0,-50,50), V500, z5, tWeldGun\WObj:=wobjHsideplate;
        MoveL offs(SP_HPivRND_PJ_Zs,150,-150,50), V500, z10, tWeldGun\WObj:=wobjHsideplate;
        MoveL offs(SP_HPivRND_PJ_Ys,150,-450,50), V500, z10, tWeldGun\WObj:=wobjHsideplate;
        MoveL offs(SP_HPivRND_PJ_Ys,150,50,50), v400, z10, tWeldGun\WObj:=wobjHsideplate;
        MoveL offs(SP_HPivRND_PJ_Ys,0,25,50), v400, z10, tWeldGun\WObj:=wobjHsideplate;
        Search_1D SR_Piv_Y\SearchStop:=PivFOUND_Y, SP_HPivRND_PJ_Ys, SP_HPivRND_PJ_Ye, v300, tWeldGun\WObj:=wobjHsideplate\SchSpeed:=10;
  		MoveL PivFOUND_Y, V500, z1, tWeldGun\WObj:=wobjHsideplate;
        WaitTime\InPos, 1;
        PivFOUND_Y := CRobT(\Tool:=tWeldgun\WObj:=obSTN1);
        WaitTime\InPos, 1;
        MoveL offs(SP_HPivRND_PJ_Ys,0,25,50), v400, z10, tWeldGun\WObj:=wobjHsideplate;
        MoveL offs(SP_HPivRND_PJ_Ys,150,50,50), v400, z10, tWeldGun\WObj:=wobjHsideplate;
        MoveL offs(SP_HPivRND_PJ_Ys,150,-450,50), V500, z10, tWeldGun\WObj:=wobjHsideplate;
        PivWobj_Translation_Locator wobj_PivCam, PivFOUND_Y, PivFOUND_Z, WPIVOTANGLE;
        WaitTime\InPos, 1;
        MoveJ offs(SP_HPivRND_PJ_Zs,150,-250,50), V500, z5, tWeldGun\WObj:=wobjHsideplate;
        MoveL offs(SP_HPivRND_PJ_Zs,-150,-250,50), V500, z5, tWeldGun\WObj:=wobjHsideplate;
        MoveJ offs(H_PJRnd_1st_s,-150, -200, -50), V500, z10, tWeldGun\WObj:=wobj_PivCam;
        MoveL offs(H_PJRnd_1st_s,-100, -150, 0), V500, z5, tWeldGun\WObj:=wobj_PivCam;
     	MoveL RelTool(SP_HRND_PJEDGE_S,0,0,-20), v100, z1, tWeldGun\WObj:=wobj_PivCam;
		Search_Edge\TopCornerDisp:=SRH_PJ_EDGE, SP_Hrnd_PjEDGE_S, SP_Hrnd_PjEDGE_E, edgedata_HRND_PJ\InitSchL:=15\Spacing:=3\PackStart, v50, tWeldGun\WObj:=wobj_PivCam\SrchSpeed:=5;
        TPWrite "SRH_PJ_EDGE XYZ:="\Pos:=SRH_PJ_EDGE.trans;
        MoveL RelTool(SP_Hrnd_PJEDGE_S,0,0,-20), v100, z1, tWeldGun\WObj:=wobj_PivCam;
		Search_Joint SRH_PJ_JOINT, SP_Hrnd_PjJOINT_S, SP_Hrnd_PjJOINT_E, bevelparam_HRND_PJ, seampar_HRND_PJ\InitSchL:=15\PackStart, v50, tWeldGun\WObj:=wobj_PivCam\PrePDisp:=SRH_PJ_EDGE\SrchSpeed:=5;
		MoveL Offs(H_PJRnd_2nd_S,-50,-75,-10), vExtMax, z1, tWeldGun\WObj:=wobj_PivCam;
        TPWrite "SRH_PJ_JOINT XYZ:="\Pos:=SRH_PJ_JOINT.trans;
        TPWrite "mm2 Weld Area Calculated:="\num:=seampar_HRND_PJ.Area;
        SRH_PJ_EDGE.trans.x := 0;
        SRH_PJ_JOINT.trans.x := 0;
        TPWrite "NOW WORKING ON WELD 'HPJ_ROUND'(root)";
        seampar_HRND_PJ.Weldpar.fill_pct := percentrootpass;
	   IF bWO455only = TRUE OR bWO456only = TRUE THEN   seampar_HRND_PJ.Weldpar.wirefeed:=(wdGH_RND_PJ_CVR.main_arc.wirefeed *60)/25.4;
	    ENDIF
	    IF bWO458only = TRUE OR bWO459only = TRUE THEN   seampar_HRND_PJ.Weldpar.wirefeed:=wdGH_RND_PJ_CVR.main_arc.wirefeed;
	    ENDIF
	    PDispSet SRH_PJ_EDGE;
		HWeldStart H_PJRnd_1st_E, seampar_HRND_PJ, smGH_RND_PJ, wdGH_RND_PJ_CVR\Weave:=wv0, v100, z1, tWeldGun\WObj:=wobj_PivCam;
		HWeldL H_PJRnd_1st_EM, seampar_HRND_PJ, v100, z1, tWeldGun\WObj:=wobj_PivCam;
        HWeldLEnd H_PJRnd_1st_s, seampar_HRND_PJ, v100, z1, tWeldGun\WObj:=wobj_PivCam;
        MoveL Offs(H_PJRnd_2nd_S,-50,-75,-10), vExtMax, z1, tWeldGun\WObj:=wobj_PivCam;
		PDispOff;
        TPWrite "NOW WORKING ON WELD 'HPJ_ROUND'(2nd pass)";
		WaitTime 4;
    	seampar_HRND_PJ.Weldpar.fill_pct := percentcoverpass;
	   IF bWO455only = TRUE OR bWO456only = TRUE THEN   seampar_HRND_PJ.Weldpar.wirefeed:=(wdGH_RND_PJ_CVR.main_arc.wirefeed *60)/25.4;
	    ENDIF
	    IF bWO458only = TRUE OR bWO459only = TRUE THEN   seampar_HRND_PJ.Weldpar.wirefeed:=wdGH_RND_PJ_CVR.main_arc.wirefeed;
	    ENDIF
		PDispSet SRH_PJ_JOINT;
		HWeldStart H_PJRnd_2nd_S, seampar_HRND_PJ, smGH_RND_PJ, wdGH_RND_PJ_CVR\Weave:=wvGH_RND_PJ_CVR, v100, z1, tWeldGun\WObj:=wobj_PivCam\Track:=trPJhiteonly1;
		HWeldL H_PJRnd_2nd_SM, seampar_HRND_PJ, v100, z1, tWeldGun\WObj:=wobj_PivCam;
		HWeldL H_PJRnd_2nd_EM, seampar_HRND_PJ, v100, z1, tWeldGun\WObj:=wobj_PivCam;
        HWeldLEnd H_PJRnd_2nd_E, seampar_HRND_PJ, v100, z1, tWeldGun\WObj:=wobj_PivCam;
		MoveL Offs(H_PJRnd_2nd_S,-50,-75,-10), vExtMax, z1, tWeldGun\WObj:=wobj_PivCam;
        MoveL offs(H_PJRnd_1st_s,-75, -150, 50), V500, z10, tWeldGun\WObj:=wobj_PivCam;
        MoveL offs(H_PJRnd_1st_s,-450, -150, 50), V500, z10, tWeldGun\WObj:=wobj_PivCam;
        MoveJ pjthomeSTA1zero, vCellSpeed, fine, tWeldGun\WObj:=wobj0;
		GOTO DONE_WELDING_PJ;
	    DONE_WELDING_PJ:
    ENDPROC

    PROC SET_PivX_Srch(INOUT
            NUM yy_SRCH_Target,
            NUM zz_SRCH_Target)

            VAR num g_H_sideplateDIST;

            IF PIVOT_USED =  674961 or PIVOT_USED =  350404 THEN  !77F - 120F CAM
                   g_H_sideplateDIST := (292.0/2) ;
           ELSEIF PIVOT_USED =  6099018 THEN  !18H CAM
                   g_H_sideplateDIST := (190.6/2) ;
           ELSEIF PIVOT_USED =  6089330 THEN  !33H RND
                   g_H_sideplateDIST := (268.0/2) ;
           ELSEIF PIVOT_USED =  6802774 THEN  !24H RND
                   g_H_sideplateDIST := (215.0/2) ;
           ELSEIF PIVOT_USED =  6870131 THEN  !34H RND
                   g_H_sideplateDIST := (279.0/2) ;
            ELSEIF PIVOT_USED = 6845931 THEN !42H RND
                   g_H_sideplateDIST := (287.0/2) ;
           ENDIF

           WaitTime\iNpOS, .1;


